Yaskawa INFORM job: DEMO_ROOF_SIDE_0625_3PAINT_28.JBI

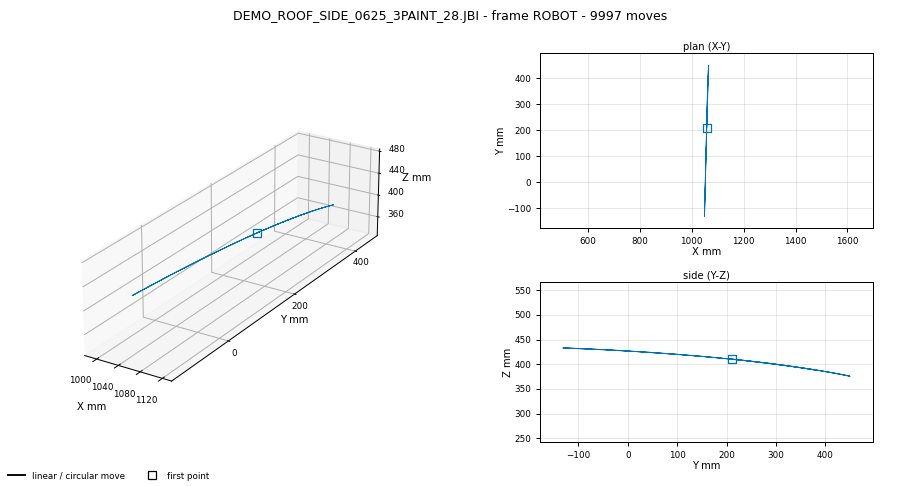
[picture p0: tool path of DEMO_ROOF_SIDE_0625_3PAINT_28.JBI in frame ROBOT, 9997 of 9997 moves have a stored position in this frame; points joined in program order, loops and branches not executed]
/JOB
//NAME DEMO_ROOF_SIDE_0625_3PAINT28
//POS
///NPOS 9997,0,0,0,0,0
///TOOL 0
///USER 0
///POSTYPE ROBOT
///RECTAN
///RCONF 1,0,0,0,0,0,0,0,0,0,0,0,0,0,0,0,0,0,0,0,0,0,0,0
C00000=1058.658,210.851,410.798,172.512,33.168,156.167
C00001=1058.665,211.100,410.772,172.514,33.173,156.168
C00002=1058.671,211.349,410.746,172.516,33.176,156.168
C00003=1058.677,211.597,410.720,172.518,33.181,156.169
C00004=1058.683,211.846,410.694,172.520,33.184,156.170
C00005=1058.690,212.094,410.668,172.522,33.189,156.171
C00006=1058.695,212.343,410.642,172.524,33.192,156.171
C00007=1058.702,212.591,410.616,172.526,33.196,156.172
C00008=1058.708,212.840,410.590,172.528,33.200,156.173
C00009=1058.714,213.088,410.564,172.530,33.204,156.174
C00010=1058.721,213.337,410.539,172.531,33.208,156.174
C00011=1058.726,213.585,410.512,172.533,33.212,156.175
C00012=1058.733,213.834,410.487,172.535,33.216,156.176
C00013=1058.738,214.082,410.460,172.537,33.220,156.177
C00014=1058.745,214.331,410.435,172.539,33.224,156.177
C00015=1058.751,214.580,410.408,172.541,33.227,156.178
C00016=1058.759,214.908,410.373,172.544,33.233,156.179
C00017=1058.767,215.238,410.338,172.546,33.238,156.180
C00018=1058.775,215.566,410.304,172.549,33.243,156.181
C00019=1058.783,215.895,410.269,172.553,33.248,156.182
C00020=1058.789,216.144,410.244,172.555,33.253,156.183
C00021=1058.795,216.392,410.217,172.557,33.256,156.184
C00022=1058.802,216.641,410.190,172.559,33.260,156.184
C00023=1058.808,216.890,410.165,172.561,33.264,156.185
C00024=1058.814,217.138,410.138,172.563,33.268,156.186
C00025=1058.820,217.386,410.112,172.565,33.271,156.186
C00026=1058.827,217.636,410.086,172.567,33.276,156.187
C00027=1058.832,217.884,410.059,172.569,33.279,156.188
C00028=1058.839,218.132,410.033,172.571,33.284,156.189
C00029=1058.845,218.380,410.007,172.573,33.287,156.189
C00030=1058.851,218.630,409.981,172.575,33.291,156.190
C00031=1058.857,218.878,409.954,172.577,33.295,156.191
C00032=1058.864,219.126,409.928,172.579,33.299,156.192
C00033=1058.870,219.375,409.901,172.581,33.302,156.192
C00034=1058.876,219.624,409.875,172.583,33.307,156.193
C00035=1058.882,219.872,409.849,172.585,33.310,156.194
C00036=1058.888,220.121,409.823,172.587,33.314,156.194
C00037=1058.895,220.369,409.796,172.589,33.318,156.195
C00038=1058.901,220.618,409.770,172.591,33.322,156.196
C00039=1058.907,220.866,409.744,172.593,33.326,156.197
C00040=1058.914,221.102,409.718,172.595,33.329,156.197
C00041=1058.918,221.337,409.693,172.598,33.333,156.198
C00042=1058.925,221.573,409.667,172.600,33.337,156.199
C00043=1058.930,221.809,409.643,172.601,33.340,156.199
C00044=1058.936,222.045,409.618,172.603,33.344,156.200
C00045=1058.942,222.280,409.593,172.605,33.348,156.201
C00046=1058.948,222.516,409.567,172.607,33.351,156.202
C00047=1058.954,222.752,409.542,172.609,33.355,156.202
C00048=1058.959,223.000,409.515,172.611,33.359,156.203
C00049=1058.966,223.249,409.488,172.613,33.363,156.204
C00050=1058.972,223.498,409.462,172.615,33.367,156.205
C00051=1058.977,223.746,409.435,172.617,33.371,156.205
C00052=1058.985,223.995,409.409,172.619,33.374,156.206
C00053=1058.990,224.243,409.382,172.621,33.379,156.207
C00054=1058.996,224.491,409.355,172.623,33.382,156.207
C00055=1059.003,224.740,409.328,172.626,33.386,156.208
C00056=1059.009,224.988,409.301,172.628,33.390,156.209
C00057=1059.016,225.237,409.275,172.630,33.394,156.210
C00058=1059.021,225.485,409.248,172.632,33.397,156.210
C00059=1059.027,225.734,409.221,172.635,33.402,156.211
C00060=1059.034,225.983,409.194,172.637,33.405,156.212
C00061=1059.039,226.231,409.168,172.639,33.409,156.212
C00062=1059.045,226.479,409.141,172.641,33.413,156.213
C00063=1059.053,226.728,409.114,172.643,33.417,156.214
C00064=1059.058,226.976,409.087,172.645,33.421,156.215
C00065=1059.065,227.225,409.060,172.647,33.424,156.215
C00066=1059.070,227.473,409.034,172.649,33.428,156.216
C00067=1059.077,227.722,409.007,172.651,33.432,156.217
C00068=1059.083,227.970,408.979,172.654,33.436,156.218
C00069=1059.090,228.219,408.953,172.656,33.439,156.218
C00070=1059.096,228.467,408.926,172.658,33.444,156.219
C00071=1059.102,228.716,408.899,172.660,33.447,156.220
C00072=1059.108,228.964,408.872,172.662,33.451,156.220
C00073=1059.114,229.212,408.845,172.664,33.455,156.221
C00074=1059.120,229.461,408.818,172.666,33.459,156.222
C00075=1059.126,229.710,408.791,172.669,33.463,156.223
C00076=1059.133,229.958,408.764,172.671,33.466,156.223
C00077=1059.139,230.207,408.737,172.673,33.470,156.224
C00078=1059.145,230.456,408.710,172.676,33.474,156.225
C00079=1059.151,230.703,408.683,172.678,33.478,156.226
C00080=1059.157,230.952,408.656,172.680,33.482,156.226
C00081=1059.164,231.200,408.628,172.682,33.486,156.227
C00082=1059.170,231.449,408.601,172.684,33.489,156.228
C00083=1059.176,231.698,408.575,172.686,33.494,156.229
C00084=1059.182,231.946,408.547,172.688,33.497,156.229
C00085=1059.188,232.194,408.520,172.690,33.501,156.230
C00086=1059.194,232.443,408.492,172.693,33.505,156.231
C00087=1059.200,232.692,408.465,172.695,33.509,156.231
C00088=1059.207,232.940,408.438,172.697,33.512,156.232
C00089=1059.212,233.188,408.411,172.700,33.516,156.233
C00090=1059.219,233.437,408.383,172.702,33.520,156.234
C00091=1059.225,233.685,408.357,172.704,33.524,156.234
C00092=1059.231,233.934,408.329,172.706,33.528,156.235
C00093=1059.236,234.182,408.302,172.708,33.532,156.236
C00094=1059.243,234.431,408.274,172.711,33.536,156.237
C00095=1059.249,234.679,408.247,172.713,33.539,156.237
C00096=1059.255,234.911,408.221,172.715,33.543,156.238
C00097=1059.261,235.142,408.196,172.717,33.546,156.239
C00098=1059.266,235.375,408.170,172.719,33.550,156.239
C00099=1059.272,235.606,408.144,172.721,33.554,156.240
C00100=1059.278,235.838,408.119,172.723,33.557,156.241
C00101=1059.284,236.070,408.093,172.725,33.560,156.241
C00102=1059.290,236.301,408.068,172.728,33.564,156.242
C00103=1059.295,236.532,408.042,172.730,33.568,156.243
C00104=1059.301,236.782,408.015,172.732,33.571,156.243
C00105=1059.307,237.030,407.987,172.734,33.576,156.244
C00106=1059.314,237.278,407.959,172.736,33.579,156.245
C00107=1059.320,237.527,407.932,172.739,33.583,156.246
C00108=1059.325,237.775,407.904,172.741,33.587,156.246
C00109=1059.332,238.023,407.877,172.743,33.591,156.247
C00110=1059.339,238.272,407.849,172.745,33.594,156.248
C00111=1059.344,238.520,407.822,172.747,33.598,156.248
C00112=1059.350,238.769,407.794,172.750,33.602,156.249
C00113=1059.357,239.017,407.766,172.752,33.606,156.250
C00114=1059.363,239.265,407.739,172.755,33.610,156.251
C00115=1059.370,239.514,407.711,172.757,33.613,156.251
C00116=1059.375,239.763,407.684,172.759,33.617,156.252
C00117=1059.382,240.011,407.656,172.762,33.621,156.253
C00118=1059.388,240.259,407.628,172.764,33.625,156.254
C00119=1059.394,240.508,407.600,172.766,33.628,156.254
C00120=1059.400,240.756,407.573,172.768,33.632,156.255
C00121=1059.407,241.004,407.545,172.770,33.636,156.256
C00122=1059.413,241.253,407.517,172.773,33.640,156.256
C00123=1059.419,241.501,407.490,172.775,33.644,156.257
C00124=1059.425,241.750,407.462,172.777,33.647,156.258
C00125=1059.431,241.998,407.434,172.780,33.651,156.259
C00126=1059.437,242.246,407.407,172.783,33.655,156.259
C00127=1059.443,242.495,407.378,172.785,33.659,156.260
C00128=1059.450,242.743,407.351,172.787,33.662,156.261
C00129=1059.455,242.991,407.323,172.789,33.666,156.261
C00130=1059.462,243.240,407.295,172.791,33.670,156.262
C00131=1059.468,243.489,407.267,172.794,33.674,156.263
C00132=1059.475,243.737,407.239,172.796,33.678,156.264
C00133=1059.480,243.985,407.211,172.798,33.682,156.265
C00134=1059.487,244.234,407.183,172.800,33.685,156.265
C00135=1059.493,244.482,407.155,172.803,33.689,156.266
C00136=1059.498,244.730,407.126,172.806,33.693,156.267
C00137=1059.505,244.978,407.098,172.808,33.697,156.267
C00138=1059.511,245.227,407.070,172.810,33.701,156.268
C00139=1059.517,245.475,407.042,172.813,33.704,156.269
C00140=1059.523,245.723,407.014,172.815,33.708,156.270
C00141=1059.530,245.972,406.987,172.817,33.712,156.270
C00142=1059.535,246.221,406.958,172.819,33.716,156.271
C00143=1059.542,246.469,406.929,172.822,33.719,156.272
C00144=1059.547,246.717,406.901,172.824,33.724,156.273
C00145=1059.554,246.965,406.874,172.826,33.727,156.273
C00146=1059.560,247.214,406.845,172.829,33.731,156.274
C00147=1059.566,247.463,406.817,172.832,33.735,156.275
C00148=1059.571,247.710,406.788,172.834,33.739,156.275
C00149=1059.578,247.959,406.761,172.836,33.743,156.276
C00150=1059.584,248.207,406.732,172.839,33.747,156.277
C00151=1059.590,248.456,406.703,172.841,33.750,156.278
C00152=1059.595,248.684,406.677,172.843,33.754,156.278
C00153=1059.601,248.913,406.652,172.845,33.757,156.279
C00154=1059.607,249.142,406.625,172.847,33.761,156.280
C00155=1059.611,249.370,406.599,172.850,33.765,156.280
C00156=1059.618,249.599,406.573,172.852,33.768,156.281
C00157=1059.623,249.828,406.547,172.854,33.771,156.282
C00158=1059.629,250.057,406.521,172.857,33.775,156.282
C00159=1059.634,250.285,406.495,172.859,33.779,156.283
C00160=1059.640,250.534,406.466,172.861,33.782,156.284
C00161=1059.647,250.782,406.437,172.863,33.786,156.285
C00162=1059.653,251.030,406.409,172.866,33.790,156.285
C00163=1059.659,251.278,406.380,172.868,33.794,156.286
C00164=1059.665,251.526,406.353,172.870,33.797,156.287
C00165=1059.671,251.774,406.323,172.873,33.802,156.288
C00166=1059.677,252.023,406.295,172.876,33.805,156.288
C00167=1059.683,252.271,406.266,172.878,33.809,156.289
C00168=1059.689,252.520,406.238,172.880,33.812,156.290
C00169=1059.695,252.768,406.209,172.883,33.817,156.291
C00170=1059.702,253.017,406.181,172.885,33.820,156.291
C00171=1059.708,253.265,406.152,172.887,33.824,156.292
C00172=1059.714,253.513,406.124,172.890,33.828,156.293
C00173=1059.720,253.761,406.095,172.893,33.832,156.293
C00174=1059.726,254.009,406.066,172.895,33.835,156.294
C00175=1059.732,254.258,406.038,172.898,33.839,156.295
C00176=1059.738,254.506,406.009,172.900,33.843,156.296
C00177=1059.745,254.754,405.981,172.903,33.847,156.296
C00178=1059.751,255.003,405.952,172.905,33.851,156.297
C00179=1059.758,255.251,405.923,172.907,33.854,156.298
C00180=1059.764,255.499,405.894,172.910,33.858,156.299
C00181=1059.770,255.748,405.865,172.912,33.862,156.299
C00182=1059.776,255.996,405.836,172.915,33.866,156.300
C00183=1059.782,256.244,405.808,172.918,33.869,156.301
C00184=1059.788,256.493,405.779,172.920,33.874,156.302
C00185=1059.794,256.741,405.750,172.922,33.877,156.302
C00186=1059.801,256.989,405.721,172.925,33.881,156.303
C00187=1059.807,257.237,405.693,172.927,33.884,156.304
C00188=1059.814,257.485,405.664,172.930,33.888,156.304
C00189=1059.820,257.734,405.635,172.932,33.892,156.305
C00190=1059.826,257.982,405.606,172.935,33.896,156.306
C00191=1059.832,258.230,405.578,172.938,33.900,156.307
C00192=1059.838,258.479,405.549,172.940,33.903,156.307
C00193=1059.845,258.727,405.520,172.943,33.907,156.308
C00194=1059.851,258.975,405.491,172.945,33.911,156.309
C00195=1059.857,259.223,405.462,172.947,33.915,156.309
C00196=1059.863,259.471,405.433,172.950,33.918,156.310
C00197=1059.869,259.720,405.404,172.952,33.922,156.311
C00198=1059.876,259.968,405.375,172.956,33.926,156.312
C00199=1059.883,260.216,405.347,172.958,33.930,156.312
C00200=1059.889,260.465,405.317,172.961,33.933,156.313
C00201=1059.896,260.713,405.288,172.963,33.937,156.314
C00202=1059.902,260.961,405.259,172.965,33.941,156.315
C00203=1059.908,261.209,405.230,172.968,33.944,156.315
C00204=1059.914,261.457,405.201,172.970,33.948,156.316
C00205=1059.921,261.705,405.172,172.973,33.952,156.317
C00206=1059.927,261.953,405.143,172.976,33.956,156.317
C00207=1059.933,262.202,405.114,172.979,33.959,156.318
C00208=1059.939,262.430,405.087,172.981,33.963,156.319
C00209=1059.945,262.657,405.060,172.983,33.966,156.319
C00210=1059.951,262.885,405.034,172.985,33.970,156.320
C00211=1059.957,263.113,405.007,172.988,33.973,156.321
C00212=1059.963,263.340,404.981,172.990,33.976,156.321
C00213=1059.968,263.568,404.954,172.992,33.980,156.322
C00214=1059.974,263.796,404.927,172.995,33.983,156.323
C00215=1059.979,264.023,404.899,172.998,33.987,156.324
C00216=1059.985,264.271,404.870,173.000,33.991,156.324
C00217=1059.992,264.519,404.841,173.002,33.995,156.325
C00218=1059.998,264.768,404.812,173.005,33.999,156.326
C00219=1060.003,265.016,404.782,173.007,34.002,156.326
C00220=1060.010,265.265,404.753,173.010,34.006,156.327
C00221=1060.017,265.512,404.723,173.013,34.010,156.328
C00222=1060.022,265.761,404.693,173.016,34.014,156.329
C00223=1060.029,266.009,404.664,173.018,34.017,156.329
C00224=1060.035,266.257,404.635,173.021,34.021,156.330
C00225=1060.041,266.505,404.605,173.023,34.025,156.331
C00226=1060.048,266.754,404.576,173.026,34.029,156.332
C00227=1060.054,267.002,404.547,173.028,34.033,156.332
C00228=1060.060,267.250,404.516,173.032,34.036,156.333
C00229=1060.066,267.498,404.487,173.034,34.040,156.334
C00230=1060.072,267.746,404.458,173.037,34.044,156.335
C00231=1060.079,267.994,404.428,173.039,34.048,156.335
C00232=1060.085,268.243,404.398,173.042,34.052,156.336
C00233=1060.091,268.491,404.369,173.044,34.055,156.337
C00234=1060.097,268.739,404.339,173.047,34.059,156.338
C00235=1060.103,268.987,404.310,173.050,34.063,156.338
C00236=1060.110,269.235,404.280,173.053,34.067,156.339
C00237=1060.116,269.483,404.250,173.055,34.071,156.340
C00238=1060.122,269.731,404.220,173.058,34.074,156.341
C00239=1060.128,269.979,404.191,173.060,34.079,156.341
C00240=1060.135,270.227,404.161,173.063,34.082,156.342
C00241=1060.141,270.476,404.131,173.065,34.086,156.343
C00242=1060.147,270.723,404.101,173.069,34.090,156.344
C00243=1060.153,270.972,404.072,173.071,34.094,156.344
C00244=1060.160,271.220,404.042,173.074,34.097,156.345
C00245=1060.165,271.469,404.012,173.076,34.101,156.346
C00246=1060.172,271.716,403.982,173.079,34.105,156.347
C00247=1060.178,271.965,403.952,173.081,34.109,156.347
C00248=1060.184,272.213,403.922,173.085,34.113,156.348
C00249=1060.190,272.461,403.892,173.087,34.116,156.349
C00250=1060.197,272.709,403.863,173.090,34.120,156.350
C00251=1060.203,272.957,403.832,173.092,34.124,156.350
C00252=1060.210,273.205,403.802,173.095,34.128,156.351
C00253=1060.215,273.453,403.773,173.097,34.132,156.352
C00254=1060.221,273.702,403.742,173.101,34.136,156.353
C00255=1060.228,273.949,403.712,173.104,34.139,156.353
C00256=1060.234,274.198,403.683,173.106,34.143,156.354
C00257=1060.240,274.446,403.652,173.109,34.147,156.355
C00258=1060.247,274.694,403.622,173.111,34.151,156.356
C00259=1060.252,274.941,403.592,173.114,34.155,156.356
C00260=1060.258,275.191,403.562,173.116,34.158,156.357
C00261=1060.265,275.438,403.532,173.120,34.163,156.358
C00262=1060.271,275.686,403.502,173.123,34.166,156.359
C00263=1060.277,275.934,403.471,173.125,34.170,156.360
C00264=1060.284,276.164,403.443,173.127,34.174,156.360
C00265=1060.289,276.394,403.416,173.130,34.178,156.361
C00266=1060.295,276.623,403.388,173.132,34.181,156.362
C00267=1060.300,276.852,403.360,173.136,34.184,156.362
C00268=1060.306,277.082,403.331,173.138,34.188,156.363
C00269=1060.311,277.312,403.304,173.140,34.191,156.364
C00270=1060.317,277.541,403.276,173.143,34.195,156.364
C00271=1060.323,277.771,403.247,173.145,34.199,156.365
C00272=1060.330,278.019,403.217,173.148,34.203,156.366
C00273=1060.336,278.266,403.187,173.151,34.206,156.367
C00274=1060.342,278.515,403.156,173.154,34.211,156.367
C00275=1060.348,278.763,403.126,173.157,34.214,156.368
C00276=1060.355,279.011,403.096,173.159,34.218,156.369
C00277=1060.361,279.259,403.065,173.162,34.222,156.370
C00278=1060.367,279.507,403.035,173.165,34.226,156.370
C00279=1060.373,279.755,403.004,173.168,34.230,156.371
C00280=1060.380,280.003,402.974,173.171,34.233,156.372
C00281=1060.386,280.251,402.944,173.173,34.237,156.373
C00282=1060.392,280.499,402.914,173.176,34.241,156.374
C00283=1060.398,280.748,402.883,173.179,34.245,156.374
C00284=1060.404,280.995,402.853,173.181,34.249,156.375
C00285=1060.411,281.243,402.821,173.185,34.253,156.376
C00286=1060.417,281.491,402.791,173.187,34.257,156.377
C00287=1060.423,281.740,402.760,173.190,34.261,156.377
C00288=1060.429,281.987,402.730,173.193,34.264,156.378
C00289=1060.435,282.236,402.699,173.195,34.269,156.379
C00290=1060.442,282.483,402.668,173.199,34.272,156.380
C00291=1060.448,282.732,402.637,173.202,34.276,156.381
C00292=1060.454,282.979,402.607,173.204,34.280,156.381
C00293=1060.460,283.228,402.576,173.207,34.284,156.382
C00294=1060.466,283.475,402.545,173.210,34.288,156.383
C00295=1060.473,283.724,402.514,173.213,34.292,156.384
C00296=1060.479,283.972,402.484,173.216,34.296,156.384
C00297=1060.485,284.219,402.453,173.219,34.300,156.385
C00298=1060.491,284.467,402.422,173.221,34.304,156.386
C00299=1060.498,284.716,402.391,173.224,34.307,156.387
C00300=1060.504,284.963,402.360,173.227,34.312,156.388
C00301=1060.510,285.212,402.330,173.230,34.315,156.388
C00302=1060.517,285.459,402.298,173.233,34.319,156.389
C00303=1060.523,285.707,402.268,173.236,34.323,156.390
C00304=1060.529,285.956,402.237,173.238,34.327,156.391
C00305=1060.535,286.203,402.206,173.241,34.331,156.391
C00306=1060.542,286.451,402.175,173.245,34.335,156.392
C00307=1060.548,286.699,402.144,173.247,34.338,156.393
C00308=1060.554,286.947,402.114,173.250,34.343,156.394
C00309=1060.561,287.195,402.082,173.253,34.347,156.395
C00310=1060.567,287.444,402.051,173.256,34.350,156.395
C00311=1060.573,287.691,402.020,173.259,34.355,156.396
C00312=1060.580,287.939,401.990,173.262,34.358,156.397
C00313=1060.587,288.187,401.958,173.265,34.362,156.398
C00314=1060.592,288.435,401.927,173.267,34.366,156.398
C00315=1060.598,288.683,401.896,173.270,34.370,156.399
C00316=1060.604,288.930,401.865,173.274,34.374,156.400
C00317=1060.611,289.179,401.834,173.277,34.378,156.401
C00318=1060.618,289.427,401.803,173.279,34.382,156.402
C00319=1060.623,289.674,401.771,173.282,34.386,156.402
C00320=1060.629,289.910,401.742,173.285,34.390,156.403
C00321=1060.636,290.145,401.712,173.288,34.393,156.404
C00322=1060.641,290.380,401.683,173.291,34.397,156.405
C00323=1060.647,290.615,401.653,173.293,34.401,156.405
C00324=1060.653,290.850,401.623,173.296,34.405,156.406
C00325=1060.659,291.084,401.594,173.299,34.408,156.407
C00326=1060.665,291.320,401.563,173.302,34.412,156.408
C00327=1060.671,291.555,401.534,173.305,34.416,156.408
C00328=1060.677,291.802,401.503,173.308,34.420,156.409
C00329=1060.683,292.050,401.471,173.310,34.424,156.410
C00330=1060.690,292.298,401.440,173.313,34.428,156.411
C00331=1060.697,292.546,401.408,173.317,34.432,156.412
C00332=1060.702,292.794,401.377,173.320,34.436,156.412
C00333=1060.709,293.042,401.345,173.322,34.440,156.413
C00334=1060.715,293.290,401.315,173.325,34.444,156.414
C00335=1060.721,293.538,401.283,173.328,34.447,156.415
C00336=1060.727,293.786,401.252,173.332,34.452,156.416
C00337=1060.734,294.033,401.220,173.335,34.456,156.416
C00338=1060.740,294.282,401.188,173.337,34.459,156.417
C00339=1060.747,294.530,401.157,173.340,34.463,156.418
C00340=1060.753,294.777,401.126,173.344,34.468,156.419
C00341=1060.759,295.025,401.094,173.347,34.472,156.420
C00342=1060.765,295.273,401.062,173.350,34.475,156.420
C00343=1060.771,295.521,401.030,173.352,34.479,156.421
C00344=1060.778,295.769,400.999,173.355,34.484,156.422
C00345=1060.784,296.017,400.967,173.359,34.488,156.423
C00346=1060.790,296.264,400.936,173.362,34.491,156.424
C00347=1060.796,296.513,400.904,173.365,34.495,156.425
C00348=1060.803,296.760,400.871,173.367,34.500,156.425
C00349=1060.809,297.008,400.839,173.371,34.504,156.426
C00350=1060.815,297.255,400.808,173.374,34.508,156.427
C00351=1060.821,297.504,400.776,173.377,34.512,156.428
C00352=1060.827,297.752,400.744,173.380,34.516,156.429
C00353=1060.834,297.999,400.712,173.382,34.520,156.429
C00354=1060.840,298.247,400.680,173.386,34.524,156.430
C00355=1060.846,298.495,400.648,173.389,34.528,156.431
C00356=1060.852,298.743,400.616,173.392,34.532,156.432
C00357=1060.859,298.990,400.584,173.395,34.536,156.433
C00358=1060.865,299.238,400.552,173.399,34.540,156.434
C00359=1060.871,299.487,400.520,173.401,34.545,156.435
C00360=1060.877,299.734,400.487,173.404,34.549,156.435
C00361=1060.883,299.981,400.456,173.407,34.553,156.436
C00362=1060.889,300.230,400.424,173.411,34.557,156.437
C00363=1060.895,300.477,400.392,173.414,34.561,156.438
C00364=1060.901,300.725,400.360,173.417,34.565,156.439
C00365=1060.908,300.973,400.327,173.419,34.569,156.440
C00366=1060.915,301.221,400.295,173.423,34.574,156.440
C00367=1060.920,301.469,400.263,173.426,34.578,156.441
C00368=1060.927,301.717,400.231,173.429,34.582,156.442
C00369=1060.932,301.964,400.199,173.432,34.586,156.443
C00370=1060.938,302.212,400.166,173.436,34.590,156.444
C00371=1060.945,302.460,400.135,173.439,34.594,156.445
C00372=1060.951,302.707,400.102,173.441,34.598,156.445
C00373=1060.958,302.955,400.069,173.444,34.602,156.446
C00374=1060.964,303.203,400.037,173.448,34.607,156.447
C00375=1060.970,303.451,400.005,173.451,34.611,156.448
C00376=1060.977,303.693,399.974,173.454,34.615,156.449
C00377=1060.983,303.936,399.942,173.457,34.618,156.450
C00378=1060.989,304.178,399.910,173.460,34.623,156.450
C00379=1060.995,304.421,399.878,173.464,34.627,156.451
C00380=1061.001,304.664,399.847,173.466,34.631,156.452
C00381=1061.007,304.906,399.815,173.469,34.635,156.453
C00382=1061.013,305.149,399.783,173.473,34.639,156.454
C00383=1061.019,305.392,399.752,173.476,34.643,156.455
C00384=1061.026,305.639,399.719,173.479,34.647,156.456
C00385=1061.033,305.887,399.687,173.482,34.651,156.456
C00386=1061.039,306.135,399.654,173.486,34.656,156.457
C00387=1061.045,306.383,399.622,173.489,34.660,156.458
C00388=1061.051,306.630,399.589,173.492,34.664,156.459
C00389=1061.058,306.878,399.556,173.495,34.668,156.460
C00390=1061.064,307.126,399.523,173.499,34.672,156.461
C00391=1061.071,307.374,399.491,173.502,34.676,156.461
C00392=1061.077,307.622,399.459,173.504,34.680,156.462
C00393=1061.084,307.869,399.426,173.507,34.684,156.463
C00394=1061.090,308.117,399.394,173.511,34.689,156.464
C00395=1061.096,308.364,399.361,173.514,34.693,156.465
C00396=1061.103,308.612,399.328,173.517,34.697,156.466
C00397=1061.109,308.860,399.295,173.520,34.701,156.467
C00398=1061.116,309.108,399.262,173.524,34.705,156.467
C00399=1061.123,309.355,399.230,173.527,34.709,156.468
C00400=1061.129,309.603,399.197,173.530,34.713,156.469
C00401=1061.135,309.850,399.165,173.533,34.717,156.470
C00402=1061.141,310.099,399.133,173.537,34.722,156.471
C00403=1061.148,310.347,399.100,173.540,34.726,156.472
C00404=1061.155,310.595,399.067,173.543,34.730,156.473
C00405=1061.161,310.842,399.033,173.547,34.734,156.473
C00406=1061.167,311.089,399.001,173.550,34.739,156.474
C00407=1061.174,311.337,398.968,173.553,34.743,156.475
C00408=1061.181,311.585,398.935,173.556,34.747,156.476
C00409=1061.187,311.833,398.902,173.560,34.751,156.477
C00410=1061.193,312.080,398.869,173.563,34.755,156.478
C00411=1061.200,312.328,398.836,173.566,34.759,156.479
C00412=1061.207,312.576,398.804,173.570,34.764,156.480
C00413=1061.213,312.823,398.771,173.573,34.768,156.480
C00414=1061.220,313.072,398.738,173.576,34.772,156.481
C00415=1061.227,313.319,398.705,173.580,34.776,156.482
C00416=1061.233,313.566,398.672,173.584,34.780,156.483
C00417=1061.240,313.815,398.639,173.587,34.784,156.484
C00418=1061.246,314.062,398.606,173.590,34.789,156.485
C00419=1061.252,314.309,398.572,173.593,34.793,156.486
C00420=1061.258,314.557,398.539,173.597,34.798,156.487
C00421=1061.265,314.806,398.506,173.600,34.802,156.487
C00422=1061.271,315.053,398.472,173.603,34.807,156.488
C00423=1061.277,315.300,398.439,173.607,34.811,156.489
C00424=1061.283,315.548,398.406,173.610,34.815,156.490
C00425=1061.290,315.796,398.372,173.613,34.820,156.491
C00426=1061.296,316.044,398.339,173.617,34.824,156.492
C00427=1061.302,316.291,398.305,173.620,34.828,156.493
C00428=1061.309,316.539,398.272,173.623,34.832,156.494
C00429=1061.315,316.786,398.238,173.627,34.837,156.495
C00430=1061.321,317.034,398.205,173.630,34.841,156.496
C00431=1061.327,317.282,398.171,173.633,34.846,156.497
C00432=1061.333,317.526,398.138,173.636,34.850,156.497
C00433=1061.340,317.771,398.105,173.640,34.855,156.498
C00434=1061.345,318.015,398.072,173.643,34.859,156.499
C00435=1061.352,318.260,398.039,173.646,34.863,156.500
C00436=1061.359,318.504,398.005,173.650,34.867,156.501
C00437=1061.365,318.749,397.973,173.653,34.872,156.502
C00438=1061.371,318.994,397.939,173.656,34.876,156.503
C00439=1061.377,319.238,397.906,173.660,34.880,156.504
C00440=1061.383,319.485,397.872,173.663,34.885,156.505
C00441=1061.390,319.733,397.838,173.666,34.889,156.506
C00442=1061.396,319.981,397.805,173.671,34.894,156.507
C00443=1061.403,320.229,397.771,173.674,34.898,156.508
C00444=1061.409,320.476,397.737,173.677,34.902,156.508
C00445=1061.416,320.724,397.703,173.681,34.907,156.509
C00446=1061.422,320.972,397.670,173.684,34.911,156.510
C00447=1061.429,321.219,397.636,173.687,34.916,156.511
C00448=1061.435,321.466,397.602,173.691,34.921,156.512
C00449=1061.442,321.714,397.568,173.694,34.925,156.513
C00450=1061.447,321.962,397.535,173.697,34.929,156.514
C00451=1061.454,322.210,397.501,173.701,34.933,156.515
C00452=1061.460,322.457,397.467,173.705,34.938,156.516
C00453=1061.467,322.705,397.433,173.708,34.943,156.517
C00454=1061.474,322.952,397.399,173.711,34.947,156.518
C00455=1061.480,323.200,397.365,173.715,34.951,156.519
C00456=1061.487,323.447,397.331,173.718,34.956,156.520
C00457=1061.493,323.695,397.297,173.721,34.960,156.521
C00458=1061.499,323.944,397.263,173.726,34.965,156.522
C00459=1061.506,324.191,397.230,173.729,34.969,156.523
C00460=1061.512,324.439,397.195,173.732,34.974,156.523
C00461=1061.519,324.685,397.162,173.736,34.978,156.524
C00462=1061.525,324.933,397.127,173.739,34.983,156.525
C00463=1061.532,325.181,397.093,173.742,34.987,156.526
C00464=1061.538,325.428,397.060,173.747,34.992,156.527
C00465=1061.545,325.676,397.024,173.750,34.996,156.528
C00466=1061.552,325.923,396.991,173.754,35.001,156.529
C00467=1061.558,326.171,396.957,173.757,35.005,156.530
C00468=1061.565,326.419,396.922,173.760,35.010,156.531
C00469=1061.572,326.666,396.888,173.765,35.014,156.532
C00470=1061.578,326.914,396.854,173.768,35.019,156.533
C00471=1061.585,327.161,396.820,173.771,35.023,156.534
C00472=1061.591,327.409,396.786,173.775,35.028,156.535
C00473=1061.598,327.657,396.751,173.779,35.032,156.536
C00474=1061.605,327.904,396.717,173.782,35.037,156.537
C00475=1061.611,328.152,396.683,173.786,35.041,156.538
C00476=1061.618,328.400,396.649,173.789,35.046,156.539
C00477=1061.625,328.647,396.614,173.792,35.050,156.540
C00478=1061.631,328.894,396.580,173.797,35.055,156.541
C00479=1061.638,329.142,396.546,173.800,35.059,156.542
C00480=1061.645,329.390,396.512,173.803,35.064,156.543
C00481=1061.651,329.637,396.477,173.807,35.068,156.544
C00482=1061.658,329.885,396.442,173.811,35.073,156.545
C00483=1061.665,330.132,396.409,173.815,35.077,156.546
C00484=1061.671,330.379,396.374,173.818,35.082,156.547
C00485=1061.678,330.627,396.339,173.822,35.087,156.547
C00486=1061.685,330.875,396.304,173.826,35.091,156.548
C00487=1061.691,331.123,396.270,173.829,35.096,156.549
C00488=1061.697,331.364,396.235,173.832,35.101,156.550
C00489=1061.704,331.606,396.202,173.836,35.105,156.551
C00490=1061.710,331.847,396.168,173.840,35.110,156.552
C00491=1061.716,332.089,396.134,173.844,35.114,156.553
C00492=1061.723,332.331,396.100,173.847,35.119,156.554
C00493=1061.729,332.572,396.066,173.850,35.124,156.555
C00494=1061.735,332.814,396.033,173.854,35.128,156.556
C00495=1061.742,333.056,395.998,173.858,35.133,156.557
C00496=1061.749,333.303,395.963,173.861,35.138,156.558
C00497=1061.755,333.550,395.929,173.865,35.142,156.559
C00498=1061.762,333.798,395.894,173.869,35.147,156.560
C00499=1061.768,334.045,395.859,173.873,35.151,156.561
C00500=1061.775,334.293,395.824,173.876,35.157,156.562
C00501=1061.781,334.541,395.789,173.879,35.161,156.563
C00502=1061.788,334.788,395.753,173.884,35.166,156.564
C00503=1061.794,335.035,395.718,173.887,35.170,156.565
C00504=1061.801,335.283,395.684,173.891,35.175,156.566
C00505=1061.808,335.531,395.649,173.895,35.180,156.568
C00506=1061.814,335.778,395.614,173.898,35.185,156.569
C00507=1061.821,336.026,395.578,173.902,35.189,156.570
C00508=1061.828,336.273,395.543,173.906,35.195,156.571
C00509=1061.834,336.520,395.509,173.910,35.199,156.572
C00510=1061.841,336.767,395.473,173.913,35.204,156.573
C00511=1061.848,337.014,395.438,173.917,35.208,156.574
C00512=1061.853,337.263,395.403,173.921,35.214,156.575
C00513=1061.860,337.510,395.368,173.925,35.218,156.576
C00514=1061.867,337.757,395.333,173.929,35.223,156.577
C00515=1061.873,338.004,395.297,173.932,35.228,156.578
C00516=1061.880,338.252,395.261,173.937,35.233,156.579
C00517=1061.887,338.499,395.226,173.940,35.238,156.580
C00518=1061.893,338.747,395.191,173.943,35.243,156.581
C00519=1061.900,338.994,395.155,173.948,35.248,156.582
C00520=1061.906,339.241,395.120,173.951,35.253,156.583
C00521=1061.913,339.489,395.085,173.956,35.257,156.584
C00522=1061.919,339.737,395.049,173.959,35.262,156.585
C00523=1061.926,339.984,395.014,173.962,35.267,156.586
C00524=1061.934,340.231,394.978,173.967,35.272,156.587
C00525=1061.940,340.479,394.942,173.970,35.277,156.588
C00526=1061.946,340.726,394.907,173.975,35.282,156.590
C00527=1061.953,340.974,394.872,173.978,35.287,156.591
C00528=1061.959,341.221,394.836,173.982,35.292,156.592
C00529=1061.966,341.468,394.800,173.986,35.297,156.593
C00530=1061.972,341.716,394.765,173.990,35.301,156.594
C00531=1061.979,341.963,394.730,173.994,35.307,156.595
C00532=1061.986,342.210,394.694,173.997,35.312,156.596
C00533=1061.993,342.458,394.658,174.002,35.316,156.597
C00534=1061.999,342.706,394.623,174.005,35.322,156.598
C00535=1062.007,342.952,394.587,174.009,35.327,156.599
C00536=1062.013,343.200,394.551,174.013,35.331,156.600
C00537=1062.020,343.447,394.515,174.017,35.336,156.601
C00538=1062.026,343.695,394.479,174.021,35.342,156.603
C00539=1062.033,343.942,394.443,174.025,35.347,156.604
C00540=1062.039,344.190,394.407,174.029,35.352,156.605
C00541=1062.046,344.436,394.372,174.033,35.357,156.606
C00542=1062.052,344.684,394.336,174.037,35.362,156.607
C00543=1062.059,344.931,394.299,174.041,35.367,156.608
C00544=1062.065,345.171,394.265,174.044,35.372,156.609
C00545=1062.072,345.410,394.230,174.048,35.377,156.610
C00546=1062.079,345.649,394.195,174.052,35.382,156.611
C00547=1062.085,345.888,394.160,174.056,35.387,156.613
C00548=1062.092,346.127,394.125,174.060,35.391,156.614
C00549=1062.098,346.367,394.091,174.063,35.396,156.615
C00550=1062.104,346.606,394.056,174.068,35.402,156.616
C00551=1062.111,346.846,394.021,174.071,35.407,156.617
C00552=1062.118,347.093,393.984,174.076,35.412,156.618
C00553=1062.125,347.340,393.948,174.079,35.417,156.619
C00554=1062.131,347.588,393.912,174.084,35.422,156.620
C00555=1062.137,347.835,393.876,174.087,35.427,156.621
C00556=1062.145,348.082,393.840,174.092,35.432,156.623
C00557=1062.151,348.329,393.803,174.095,35.437,156.624
C00558=1062.157,348.576,393.767,174.100,35.443,156.625
C00559=1062.165,348.824,393.730,174.103,35.448,156.626
C00560=1062.171,349.071,393.694,174.108,35.453,156.627
C00561=1062.177,349.319,393.658,174.111,35.458,156.628
C00562=1062.184,349.566,393.621,174.116,35.464,156.629
C00563=1062.191,349.813,393.586,174.120,35.469,156.631
C00564=1062.198,350.061,393.549,174.124,35.474,156.632
C00565=1062.205,350.308,393.512,174.128,35.479,156.633
C00566=1062.211,350.555,393.476,174.132,35.484,156.634
C00567=1062.219,350.802,393.440,174.136,35.490,156.635
C00568=1062.225,351.049,393.403,174.140,35.495,156.636
C00569=1062.232,351.297,393.366,174.144,35.500,156.638
C00570=1062.239,351.544,393.329,174.149,35.505,156.639
C00571=1062.246,351.791,393.293,174.152,35.511,156.640
C00572=1062.253,352.038,393.257,174.157,35.516,156.641
C00573=1062.259,352.285,393.220,174.160,35.522,156.642
C00574=1062.266,352.533,393.183,174.165,35.527,156.643
C00575=1062.273,352.779,393.146,174.169,35.532,156.645
C00576=1062.280,353.027,393.109,174.173,35.538,156.646
C00577=1062.286,353.274,393.073,174.177,35.543,156.647
C00578=1062.293,353.521,393.035,174.182,35.548,156.648
C00579=1062.299,353.768,392.999,174.186,35.554,156.650
C00580=1062.306,354.016,392.962,174.190,35.559,156.651
C00581=1062.313,354.263,392.925,174.194,35.565,156.652
C00582=1062.320,354.510,392.888,174.198,35.570,156.653
C00583=1062.326,354.757,392.852,174.203,35.576,156.654
C00584=1062.334,355.005,392.814,174.206,35.581,156.656
C00585=1062.340,355.252,392.778,174.211,35.586,156.657
C00586=1062.347,355.499,392.740,174.215,35.592,156.658
C00587=1062.353,355.746,392.704,174.219,35.597,156.659
C00588=1062.361,355.993,392.666,174.224,35.603,156.660
C00589=1062.368,356.241,392.629,174.228,35.608,156.662
C00590=1062.374,356.487,392.592,174.232,35.613,156.663
C00591=1062.381,356.735,392.556,174.236,35.619,156.664
C00592=1062.388,356.981,392.518,174.241,35.625,156.665
C00593=1062.395,357.228,392.481,174.244,35.630,156.667
C00594=1062.402,357.476,392.444,174.249,35.635,156.668
C00595=1062.409,357.723,392.407,174.254,35.641,156.669
C00596=1062.416,357.970,392.369,174.257,35.647,156.670
C00597=1062.423,358.218,392.333,174.262,35.652,156.672
C00598=1062.430,358.464,392.295,174.266,35.657,156.673
C00599=1062.436,358.711,392.257,174.271,35.663,156.674
C00600=1062.442,358.953,392.221,174.274,35.669,156.675
C00601=1062.450,359.195,392.184,174.279,35.674,156.677
C00602=1062.456,359.436,392.148,174.284,35.680,156.678
C00603=1062.463,359.677,392.111,174.287,35.685,156.679
C00604=1062.469,359.919,392.075,174.292,35.691,156.680
C00605=1062.476,360.161,392.038,174.295,35.696,156.682
C00606=1062.483,360.402,392.001,174.300,35.702,156.683
C00607=1062.490,360.643,391.965,174.305,35.708,156.684
C00608=1062.497,360.890,391.927,174.309,35.713,156.685
C00609=1062.504,361.137,391.890,174.313,35.719,156.687
C00610=1062.510,361.384,391.852,174.317,35.725,156.688
C00611=1062.517,361.631,391.814,174.322,35.730,156.689
C00612=1062.525,361.878,391.777,174.327,35.736,156.690
C00613=1062.532,362.125,391.739,174.330,35.741,156.692
C00614=1062.538,362.373,391.701,174.335,35.748,156.693
C00615=1062.545,362.619,391.664,174.340,35.753,156.694
C00616=1062.552,362.866,391.627,174.344,35.759,156.696
C00617=1062.559,363.114,391.588,174.349,35.764,156.697
C00618=1062.566,363.360,391.550,174.353,35.771,156.698
C00619=1062.574,363.607,391.513,174.357,35.776,156.700
C00620=1062.580,363.855,391.475,174.362,35.782,156.701
C00621=1062.587,364.102,391.437,174.366,35.788,156.702
C00622=1062.593,364.349,391.399,174.371,35.794,156.704
C00623=1062.601,364.595,391.361,174.375,35.800,156.705
C00624=1062.607,364.842,391.323,174.379,35.805,156.706
C00625=1062.615,365.090,391.285,174.384,35.812,156.708
C00626=1062.621,365.336,391.247,174.389,35.817,156.709
C00627=1062.629,365.584,391.209,174.393,35.823,156.710
C00628=1062.635,365.830,391.170,174.398,35.829,156.712
C00629=1062.642,366.077,391.133,174.402,35.835,156.713
C00630=1062.649,366.324,391.094,174.406,35.841,156.715
C00631=1062.656,366.571,391.057,174.411,35.847,156.716
C00632=1062.663,366.818,391.018,174.416,35.853,156.717
C00633=1062.669,367.065,390.980,174.420,35.859,156.719
C00634=1062.677,367.312,390.941,174.425,35.865,156.720
C00635=1062.684,367.559,390.903,174.430,35.871,156.721
C00636=1062.691,367.806,390.865,174.435,35.877,156.723
C00637=1062.698,368.052,390.826,174.438,35.883,156.724
C00638=1062.704,368.300,390.788,174.443,35.889,156.725
C00639=1062.712,368.546,390.750,174.448,35.895,156.727
C00640=1062.719,368.793,390.711,174.452,35.901,156.728
C00641=1062.726,369.040,390.673,174.457,35.907,156.730
C00642=1062.733,369.287,390.635,174.462,35.913,156.731
C00643=1062.740,369.534,390.596,174.466,35.919,156.733
C00644=1062.747,369.780,390.558,174.471,35.926,156.734
C00645=1062.754,370.027,390.519,174.476,35.932,156.735
C00646=1062.760,370.275,390.481,174.481,35.938,156.737
C00647=1062.769,370.522,390.442,174.485,35.944,156.738
C00648=1062.775,370.769,390.403,174.490,35.950,156.740
C00649=1062.783,371.015,390.365,174.495,35.956,156.741
C00650=1062.790,371.262,390.326,174.500,35.962,156.742
C00651=1062.797,371.509,390.287,174.504,35.969,156.744
C00652=1062.804,371.755,390.249,174.508,35.975,156.745
C00653=1062.811,372.002,390.210,174.513,35.981,156.747
C00654=1062.818,372.250,390.171,174.517,35.987,156.748
C00655=1062.826,372.496,390.133,174.522,35.993,156.750
C00656=1062.833,372.749,390.092,174.528,36.000,156.751
C00657=1062.840,373.004,390.052,174.533,36.006,156.752
C00658=1062.848,373.258,390.012,174.538,36.012,156.754
C00659=1062.854,373.511,389.973,174.542,36.019,156.756
C00660=1062.862,373.758,389.933,174.547,36.025,156.757
C00661=1062.868,374.005,389.894,174.552,36.032,156.759
C00662=1062.875,374.252,389.855,174.557,36.038,156.760
C00663=1062.882,374.499,389.816,174.562,36.045,156.762
C00664=1062.889,374.745,389.777,174.566,36.051,156.763
C00665=1062.897,374.993,389.738,174.571,36.057,156.765
C00666=1062.903,375.239,389.699,174.576,36.064,156.766
C00667=1062.911,375.486,389.659,174.581,36.070,156.768
C00668=1062.918,375.732,389.621,174.586,36.077,156.769
C00669=1062.926,375.979,389.581,174.590,36.083,156.770
C00670=1062.933,376.226,389.542,174.595,36.090,156.772
C00671=1062.940,376.472,389.503,174.600,36.096,156.774
C00672=1062.947,376.720,389.463,174.605,36.102,156.775
C00673=1062.954,376.966,389.424,174.610,36.109,156.777
C00674=1062.961,377.213,389.385,174.614,36.116,156.778
C00675=1062.969,377.460,389.345,174.620,36.122,156.780
C00676=1062.976,377.706,389.306,174.625,36.128,156.781
C00677=1062.983,377.953,389.267,174.630,36.135,156.783
C00678=1062.990,378.199,389.227,174.635,36.142,156.784
C00679=1062.997,378.446,389.188,174.640,36.148,156.786
C00680=1063.004,378.694,389.147,174.644,36.155,156.787
C00681=1063.011,378.940,389.108,174.649,36.162,156.789
C00682=1063.018,379.187,389.069,174.654,36.168,156.790
C00683=1063.026,379.433,389.029,174.659,36.175,156.792
C00684=1063.033,379.680,388.990,174.665,36.181,156.794
C00685=1063.041,379.927,388.950,174.670,36.188,156.795
C00686=1063.048,380.173,388.910,174.674,36.195,156.797
C00687=1063.055,380.420,388.871,174.679,36.201,156.798
C00688=1063.062,380.666,388.831,174.684,36.208,156.800
C00689=1063.070,380.913,388.791,174.689,36.215,156.801
C00690=1063.077,381.160,388.752,174.695,36.222,156.803
C00691=1063.084,381.407,388.711,174.700,36.228,156.805
C00692=1063.091,381.653,388.672,174.705,36.235,156.806
C00693=1063.099,381.900,388.632,174.710,36.242,156.808
C00694=1063.105,382.146,388.592,174.715,36.249,156.810
C00695=1063.113,382.393,388.551,174.721,36.256,156.811
C00696=1063.121,382.639,388.512,174.725,36.262,156.813
C00697=1063.128,382.886,388.471,174.730,36.270,156.814
C00698=1063.135,383.133,388.431,174.735,36.276,156.816
C00699=1063.142,383.379,388.392,174.740,36.283,156.818
C00700=1063.149,383.626,388.351,174.746,36.290,156.819
C00701=1063.157,383.872,388.311,174.751,36.297,156.821
C00702=1063.164,384.119,388.270,174.756,36.304,156.823
C00703=1063.171,384.366,388.230,174.761,36.311,156.824
C00704=1063.179,384.612,388.190,174.767,36.318,156.826
C00705=1063.186,384.859,388.150,174.772,36.325,156.828
C00706=1063.194,385.106,388.110,174.777,36.332,156.829
C00707=1063.200,385.352,388.069,174.782,36.339,156.831
C00708=1063.208,385.599,388.029,174.788,36.346,156.833
C00709=1063.216,385.845,387.988,174.793,36.353,156.834
C00710=1063.222,386.091,387.948,174.798,36.360,156.836
C00711=1063.230,386.338,387.908,174.804,36.367,156.838
C00712=1063.239,386.623,387.861,174.809,36.376,156.840
C00713=1063.248,386.907,387.814,174.815,36.384,156.842
C00714=1063.256,387.191,387.768,174.821,36.392,156.844
C00715=1063.265,387.476,387.721,174.827,36.400,156.846
C00716=1063.272,387.722,387.680,174.833,36.407,156.847
C00717=1063.280,387.969,387.640,174.838,36.414,156.849
C00718=1063.287,388.216,387.598,174.844,36.421,156.851
C00719=1063.295,388.462,387.558,174.849,36.429,156.853
C00720=1063.302,388.708,387.517,174.854,36.436,156.854
C00721=1063.310,388.955,387.477,174.860,36.443,156.856
C00722=1063.317,389.202,387.436,174.865,36.450,156.858
C00723=1063.325,389.448,387.395,174.870,36.458,156.860
C00724=1063.332,389.694,387.354,174.876,36.465,156.861
C00725=1063.340,389.941,387.313,174.881,36.472,156.863
C00726=1063.347,390.187,387.272,174.887,36.480,156.865
C00727=1063.355,390.434,387.231,174.892,36.487,156.867
C00728=1063.363,390.680,387.190,174.898,36.495,156.868
C00729=1063.370,390.927,387.149,174.904,36.502,156.870
C00730=1063.378,391.173,387.108,174.909,36.509,156.872
C00731=1063.385,391.420,387.067,174.915,36.517,156.874
C00732=1063.393,391.666,387.026,174.920,36.525,156.876
C00733=1063.401,391.913,386.985,174.926,36.532,156.877
C00734=1063.408,392.159,386.944,174.931,36.539,156.879
C00735=1063.416,392.405,386.902,174.937,36.547,156.881
C00736=1063.423,392.652,386.861,174.942,36.555,156.883
C00737=1063.431,392.898,386.820,174.948,36.562,156.885
C00738=1063.438,393.145,386.779,174.953,36.570,156.887
C00739=1063.446,393.391,386.737,174.960,36.577,156.889
C00740=1063.453,393.637,386.696,174.965,36.585,156.890
C00741=1063.461,393.883,386.654,174.970,36.593,156.892
C00742=1063.469,394.129,386.613,174.976,36.600,156.894
C00743=1063.476,394.376,386.572,174.981,36.608,156.896
C00744=1063.484,394.622,386.530,174.987,36.615,156.898
C00745=1063.491,394.869,386.489,174.993,36.623,156.900
C00746=1063.498,395.115,386.447,174.999,36.631,156.902
C00747=1063.506,395.362,386.405,175.005,36.639,156.904
C00748=1063.514,395.608,386.363,175.010,36.646,156.905
C00749=1063.521,395.854,386.321,175.016,36.654,156.907
C00750=1063.529,396.100,386.280,175.021,36.662,156.909
C00751=1063.536,396.346,386.238,175.027,36.670,156.911
C00752=1063.544,396.592,386.196,175.033,36.678,156.913
C00753=1063.552,396.840,386.155,175.039,36.686,156.915
C00754=1063.559,397.086,386.113,175.045,36.693,156.917
C00755=1063.568,397.331,386.071,175.050,36.702,156.919
C00756=1063.576,397.578,386.029,175.056,36.709,156.921
C00757=1063.583,397.825,385.987,175.062,36.717,156.923
C00758=1063.590,398.071,385.945,175.068,36.725,156.925
C00759=1063.598,398.317,385.903,175.074,36.733,156.927
C00760=1063.606,398.563,385.861,175.079,36.742,156.929
C00761=1063.613,398.809,385.819,175.086,36.750,156.931
C00762=1063.622,399.056,385.777,175.091,36.757,156.933
C00763=1063.629,399.302,385.735,175.097,36.765,156.935
C00764=1063.636,399.548,385.692,175.103,36.774,156.937
C00765=1063.644,399.795,385.650,175.109,36.782,156.939
C00766=1063.652,400.041,385.608,175.115,36.790,156.941
C00767=1063.660,400.288,385.566,175.121,36.798,156.943
C00768=1063.670,400.609,385.510,175.129,36.809,156.946
C00769=1063.681,400.931,385.455,175.137,36.820,156.948
C00770=1063.691,401.253,385.399,175.144,36.831,156.951
C00771=1063.701,401.575,385.344,175.152,36.841,156.954
C00772=1063.709,401.822,385.301,175.158,36.849,156.956
C00773=1063.716,402.068,385.259,175.165,36.858,156.958
C00774=1063.724,402.314,385.217,175.171,36.866,156.960
C00775=1063.733,402.560,385.174,175.176,36.875,156.962
C00776=1063.740,402.807,385.131,175.183,36.883,156.964
C00777=1063.748,403.053,385.088,175.189,36.891,156.966
C00778=1063.756,403.299,385.046,175.196,36.900,156.968
C00779=1063.764,403.545,385.002,175.201,36.908,156.970
C00780=1063.772,403.792,384.960,175.207,36.917,156.972
C00781=1063.779,404.037,384.917,175.214,36.925,156.975
C00782=1063.787,404.284,384.875,175.220,36.934,156.977
C00783=1063.796,404.530,384.831,175.227,36.942,156.979
C00784=1063.803,404.776,384.788,175.233,36.951,156.981
C00785=1063.811,405.022,384.745,175.238,36.959,156.983
C00786=1063.819,405.269,384.702,175.245,36.968,156.985
C00787=1063.827,405.514,384.660,175.251,36.977,156.987
C00788=1063.835,405.760,384.616,175.258,36.985,156.990
C00789=1063.843,406.006,384.573,175.264,36.994,156.992
C00790=1063.851,406.253,384.529,175.271,37.003,156.994
C00791=1063.858,406.499,384.486,175.277,37.011,156.996
C00792=1063.866,406.745,384.444,175.283,37.020,156.999
C00793=1063.874,406.992,384.400,175.289,37.029,157.001
C00794=1063.883,407.237,384.356,175.296,37.038,157.003
C00795=1063.891,407.483,384.313,175.302,37.047,157.005
C00796=1063.898,407.729,384.270,175.309,37.056,157.007
C00797=1063.906,407.975,384.227,175.315,37.065,157.010
C00798=1063.914,408.221,384.183,175.322,37.073,157.012
C00799=1063.922,408.468,384.139,175.328,37.082,157.014
C00800=1063.930,408.714,384.096,175.335,37.091,157.017
C00801=1063.938,408.960,384.052,175.341,37.101,157.019
C00802=1063.946,409.206,384.008,175.348,37.110,157.021
C00803=1063.955,409.452,383.965,175.354,37.119,157.023
C00804=1063.963,409.698,383.921,175.361,37.128,157.026
C00805=1063.970,409.944,383.877,175.367,37.137,157.028
C00806=1063.978,410.190,383.834,175.374,37.146,157.030
C00807=1063.987,410.436,383.790,175.381,37.155,157.033
C00808=1063.995,410.682,383.746,175.387,37.164,157.035
C00809=1064.003,410.928,383.702,175.394,37.173,157.037
C00810=1064.011,411.174,383.659,175.400,37.183,157.040
C00811=1064.019,411.420,383.615,175.408,37.192,157.042
C00812=1064.027,411.666,383.571,175.415,37.201,157.044
C00813=1064.035,411.912,383.527,175.421,37.210,157.047
C00814=1064.044,412.157,383.483,175.428,37.219,157.049
C00815=1064.052,412.404,383.439,175.435,37.229,157.052
C00816=1064.060,412.650,383.395,175.441,37.238,157.054
C00817=1064.068,412.896,383.350,175.448,37.247,157.056
C00818=1064.077,413.142,383.306,175.456,37.257,157.059
C00819=1064.085,413.387,383.262,175.462,37.266,157.061
C00820=1064.093,413.613,383.221,175.469,37.275,157.063
C00821=1064.101,413.838,383.181,175.474,37.283,157.066
C00822=1064.108,414.063,383.141,175.481,37.292,157.068
C00823=1064.116,414.288,383.100,175.488,37.301,157.070
C00824=1064.126,414.594,383.045,175.496,37.312,157.073
C00825=1064.136,414.900,382.990,175.505,37.325,157.076
C00826=1064.147,415.206,382.934,175.513,37.337,157.079
C00827=1064.157,415.512,382.879,175.522,37.348,157.082
C00828=1064.165,415.758,382.834,175.529,37.358,157.085
C00829=1064.173,416.003,382.789,175.537,37.368,157.087
C00830=1064.181,416.250,382.744,175.544,37.378,157.090
C00831=1064.190,416.495,382.700,175.551,37.387,157.093
C00832=1064.199,416.741,382.654,175.558,37.397,157.095
C00833=1064.207,416.987,382.610,175.565,37.407,157.098
C00834=1064.215,417.233,382.566,175.572,37.417,157.100
C00835=1064.224,417.479,382.520,175.580,37.427,157.103
C00836=1064.232,417.724,382.476,175.587,37.437,157.105
C00837=1064.241,417.970,382.430,175.594,37.447,157.108
C00838=1064.249,418.216,382.386,175.602,37.457,157.111
C00839=1064.257,418.462,382.340,175.609,37.467,157.113
C00840=1064.265,418.707,382.295,175.616,37.477,157.116
C00841=1064.274,418.954,382.250,175.623,37.487,157.119
C00842=1064.282,419.199,382.205,175.631,37.497,157.121
C00843=1064.291,419.444,382.160,175.638,37.507,157.124
C00844=1064.300,419.691,382.115,175.646,37.517,157.127
C00845=1064.308,419.936,382.070,175.653,37.527,157.129
C00846=1064.317,420.182,382.024,175.661,37.538,157.132
C00847=1064.326,420.428,381.979,175.668,37.548,157.135
C00848=1064.334,420.673,381.934,175.676,37.558,157.137
C00849=1064.342,420.919,381.888,175.683,37.568,157.140
C00850=1064.351,421.165,381.842,175.691,37.579,157.143
C00851=1064.360,421.410,381.797,175.698,37.589,157.145
C00852=1064.368,421.656,381.751,175.706,37.600,157.148
C00853=1064.377,421.902,381.706,175.713,37.610,157.151
C00854=1064.385,422.147,381.659,175.721,37.621,157.154
C00855=1064.394,422.393,381.614,175.729,37.631,157.156
C00856=1064.402,422.639,381.568,175.737,37.642,157.159
C00857=1064.411,422.885,381.523,175.745,37.652,157.162
C00858=1064.420,423.129,381.477,175.753,37.663,157.165
C00859=1064.428,423.375,381.431,175.760,37.674,157.168
C00860=1064.437,423.621,381.385,175.768,37.684,157.170
C00861=1064.445,423.867,381.339,175.776,37.695,157.173
C00862=1064.454,424.113,381.293,175.783,37.705,157.176
C00863=1064.463,424.358,381.246,175.792,37.716,157.179
C00864=1064.472,424.604,381.201,175.800,37.727,157.182
C00865=1064.480,424.849,381.154,175.808,37.738,157.185
C00866=1064.490,425.095,381.108,175.815,37.749,157.188
C00867=1064.497,425.340,381.063,175.823,37.760,157.191
C00868=1064.507,425.585,381.016,175.832,37.770,157.194
C00869=1064.515,425.831,380.970,175.840,37.781,157.196
C00870=1064.525,426.077,380.923,175.848,37.792,157.199
C00871=1064.534,426.322,380.876,175.855,37.803,157.202
C00872=1064.543,426.568,380.831,175.864,37.814,157.205
C00873=1064.551,426.814,380.784,175.872,37.825,157.208
C00874=1064.560,427.059,380.738,175.880,37.836,157.211
C00875=1064.569,427.304,380.691,175.888,37.847,157.214
C00876=1064.578,427.550,380.645,175.897,37.859,157.217
C00877=1064.586,427.795,380.598,175.905,37.870,157.220
C00878=1064.596,428.040,380.551,175.914,37.881,157.223
C00879=1064.604,428.285,380.504,175.922,37.892,157.226
C00880=1064.616,428.612,380.443,175.933,37.907,157.230
C00881=1064.627,428.938,380.380,175.943,37.923,157.235
C00882=1064.640,429.264,380.317,175.955,37.938,157.239
C00883=1064.652,429.589,380.255,175.966,37.953,157.243
C00884=1064.661,429.835,380.208,175.974,37.964,157.246
C00885=1064.670,430.080,380.160,175.984,37.976,157.249
C00886=1064.679,430.326,380.114,175.992,37.988,157.252
C00887=1064.688,430.571,380.066,176.001,37.999,157.255
C00888=1064.697,430.817,380.020,176.009,38.011,157.259
C00889=1064.706,431.062,379.972,176.018,38.022,157.262
C00890=1064.715,431.307,379.924,176.026,38.034,157.265
C00891=1064.724,431.553,379.878,176.035,38.046,157.268
C00892=1064.733,431.798,379.830,176.044,38.058,157.271
C00893=1064.742,432.043,379.782,176.052,38.070,157.275
C00894=1064.751,432.288,379.735,176.062,38.081,157.278
C00895=1064.760,432.534,379.687,176.070,38.093,157.281
C00896=1064.769,432.779,379.640,176.079,38.105,157.284
C00897=1064.779,433.024,379.592,176.088,38.118,157.288
C00898=1064.788,433.269,379.544,176.097,38.129,157.291
C00899=1064.797,433.515,379.497,176.106,38.141,157.294
C00900=1064.806,433.759,379.448,176.115,38.153,157.298
C00901=1064.816,434.004,379.401,176.124,38.166,157.301
C00902=1064.825,434.249,379.353,176.133,38.178,157.304
C00903=1064.834,434.495,379.305,176.142,38.190,157.308
C00904=1064.843,434.740,379.256,176.151,38.202,157.311
C00905=1064.852,434.985,379.209,176.161,38.215,157.314
C00906=1064.861,435.231,379.161,176.169,38.227,157.318
C00907=1064.871,435.476,379.112,176.179,38.239,157.321
C00908=1064.880,435.720,379.064,176.188,38.251,157.325
C00909=1064.890,435.966,379.017,176.197,38.264,157.328
C00910=1064.899,436.211,378.968,176.207,38.276,157.332
C00911=1064.909,436.456,378.920,176.216,38.289,157.335
C00912=1064.918,436.700,378.872,176.226,38.301,157.339
C00913=1064.927,436.946,378.823,176.234,38.314,157.342
C00914=1064.937,437.191,378.774,176.244,38.326,157.346
C00915=1064.946,437.436,378.727,176.253,38.339,157.349
C00916=1064.956,437.681,378.678,176.263,38.352,157.353
C00917=1064.966,437.926,378.629,176.273,38.365,157.356
C00918=1064.976,438.171,378.581,176.282,38.377,157.360
C00919=1064.985,438.416,378.532,176.292,38.390,157.363
C00920=1064.994,438.661,378.483,176.301,38.403,157.367
C00921=1065.004,438.906,378.433,176.312,38.416,157.371
C00922=1065.013,439.151,378.385,176.322,38.429,157.374
C00923=1065.023,439.396,378.336,176.331,38.442,157.378
C00924=1065.032,439.641,378.287,176.341,38.455,157.382
C00925=1065.042,439.886,378.238,176.351,38.468,157.385
C00926=1065.052,440.131,378.190,176.360,38.481,157.389
C00927=1065.061,440.376,378.140,176.370,38.494,157.393
C00928=1065.071,440.620,378.091,176.381,38.508,157.397
C00929=1065.080,440.865,378.041,176.391,38.521,157.400
C00930=1065.090,441.110,377.993,176.401,38.534,157.404
C00931=1065.100,441.355,377.943,176.410,38.548,157.408
C00932=1065.110,441.600,377.893,176.421,38.561,157.412
C00933=1065.119,441.845,377.844,176.431,38.574,157.416
C00934=1065.129,442.089,377.795,176.441,38.588,157.419
C00935=1065.139,442.335,377.745,176.452,38.602,157.423
C00936=1065.156,442.743,377.662,176.468,38.624,157.430
C00937=1065.172,443.152,377.579,176.486,38.647,157.436
C00938=1065.189,443.560,377.496,176.504,38.670,157.443
C00939=1065.205,443.969,377.413,176.522,38.693,157.449
C00940=1065.215,444.214,377.363,176.532,38.707,157.453
C00941=1065.225,444.458,377.313,176.543,38.721,157.457
C00942=1065.235,444.703,377.263,176.553,38.735,157.461
C00943=1065.244,444.948,377.213,176.564,38.749,157.466
C00944=1065.255,445.192,377.163,176.574,38.763,157.470
C00945=1065.265,445.437,377.113,176.585,38.777,157.474
C00946=1065.275,445.682,377.062,176.596,38.791,157.478
C00947=1065.284,445.926,377.011,176.607,38.805,157.482
C00948=1065.295,446.171,376.962,176.618,38.820,157.486
C00949=1065.305,446.415,376.911,176.629,38.834,157.490
C00950=1065.315,446.660,376.860,176.639,38.848,157.494
C00951=1065.326,446.904,376.810,176.651,38.862,157.498
C00952=1065.336,447.148,376.759,176.662,38.877,157.503
C00953=1065.346,447.392,376.709,176.673,38.891,157.507
C00954=1065.356,447.637,376.658,176.685,38.906,157.511
C00955=1065.367,447.881,376.608,176.695,38.920,157.515
C00956=1065.378,448.124,376.559,176.707,38.934,157.519
C00957=1065.391,448.368,376.510,176.718,38.948,157.524
C00958=1065.404,448.612,376.461,176.729,38.961,157.527
C00959=1065.420,448.858,376.414,176.741,38.975,157.531
C00960=1065.435,449.103,376.367,176.753,38.988,157.535
C00961=1065.452,449.347,376.320,176.764,39.000,157.539
C00962=1065.470,449.593,376.275,176.775,39.012,157.543
C00963=1065.488,449.838,376.230,176.786,39.024,157.546
C00964=1065.149,449.843,375.964,176.777,39.149,157.580
C00965=1065.130,449.598,376.009,176.766,39.138,157.577
C00966=1065.112,449.353,376.054,176.755,39.126,157.573
C00967=1065.095,449.107,376.101,176.743,39.113,157.569
C00968=1065.079,448.863,376.147,176.732,39.100,157.565
C00969=1065.064,448.617,376.195,176.720,39.087,157.561
C00970=1065.050,448.373,376.244,176.709,39.074,157.558
C00971=1065.037,448.130,376.293,176.697,39.060,157.553
C00972=1065.026,447.886,376.342,176.685,39.046,157.549
C00973=1065.015,447.642,376.392,176.674,39.032,157.545
C00974=1065.004,447.397,376.443,176.663,39.018,157.541
C00975=1064.995,447.153,376.493,176.651,39.003,157.537
C00976=1064.984,446.910,376.544,176.641,38.989,157.532
C00977=1064.974,446.666,376.595,176.629,38.974,157.528
C00978=1064.964,446.420,376.645,176.618,38.960,157.524
C00979=1064.954,446.176,376.696,176.607,38.946,157.520
C00980=1064.943,445.932,376.746,176.596,38.932,157.516
C00981=1064.933,445.687,376.797,176.585,38.918,157.512
C00982=1064.924,445.442,376.847,176.574,38.904,157.508
C00983=1064.913,445.198,376.897,176.563,38.890,157.503
C00984=1064.903,444.953,376.947,176.553,38.876,157.499
C00985=1064.893,444.709,376.998,176.542,38.862,157.495
C00986=1064.883,444.463,377.048,176.531,38.848,157.491
C00987=1064.873,444.219,377.098,176.520,38.834,157.487
C00988=1064.863,443.975,377.148,176.509,38.820,157.483
C00989=1064.848,443.585,377.227,176.492,38.798,157.477
C00990=1064.831,443.196,377.307,176.476,38.776,157.471
C00991=1064.815,442.806,377.386,176.459,38.754,157.464
C00992=1064.800,442.417,377.465,176.443,38.733,157.458
C00993=1064.790,442.172,377.515,176.432,38.719,157.454
C00994=1064.780,441.927,377.564,176.422,38.706,157.450
C00995=1064.770,441.682,377.613,176.411,38.692,157.447
C00996=1064.761,441.438,377.663,176.401,38.679,157.443
C00997=1064.750,441.193,377.713,176.391,38.666,157.439
C00998=1064.741,440.947,377.762,176.380,38.652,157.435
C00999=1064.731,440.703,377.811,176.371,38.639,157.431
C01000=1064.722,440.458,377.861,176.361,38.626,157.428
C01001=1064.712,440.213,377.909,176.351,38.613,157.424
C01002=1064.702,439.968,377.960,176.340,38.600,157.420
C01003=1064.693,439.723,378.008,176.331,38.587,157.416
C01004=1064.683,439.478,378.057,176.321,38.574,157.413
C01005=1064.673,439.233,378.106,176.311,38.561,157.409
C01006=1064.664,438.988,378.155,176.302,38.548,157.405
C01007=1064.655,438.743,378.204,176.291,38.535,157.402
C01008=1064.645,438.499,378.253,176.281,38.522,157.398
C01009=1064.635,438.254,378.302,176.272,38.509,157.395
C01010=1064.626,438.008,378.351,176.262,38.497,157.391
C01011=1064.616,437.763,378.399,176.252,38.484,157.387
C01012=1064.606,437.519,378.448,176.243,38.471,157.384
C01013=1064.597,437.274,378.497,176.233,38.458,157.380
C01014=1064.587,437.028,378.544,176.224,38.446,157.377
C01015=1064.577,436.783,378.593,176.214,38.434,157.373
C01016=1064.568,436.539,378.641,176.205,38.421,157.370
C01017=1064.559,436.293,378.690,176.195,38.409,157.366
C01018=1064.550,436.048,378.738,176.186,38.396,157.363
C01019=1064.540,435.803,378.787,176.176,38.383,157.359
C01020=1064.530,435.558,378.835,176.167,38.371,157.356
C01021=1064.521,435.313,378.882,176.157,38.359,157.352
C01022=1064.512,435.068,378.931,176.149,38.347,157.349
C01023=1064.502,434.822,378.979,176.140,38.334,157.346
C01024=1064.493,434.578,379.027,176.130,38.322,157.342
C01025=1064.484,434.333,379.075,176.121,38.310,157.339
C01026=1064.474,434.087,379.123,176.111,38.298,157.335
C01027=1064.466,433.842,379.171,176.102,38.286,157.332
C01028=1064.456,433.597,379.219,176.094,38.273,157.329
C01029=1064.447,433.351,379.267,176.085,38.262,157.325
C01030=1064.438,433.106,379.314,176.075,38.250,157.322
C01031=1064.428,432.861,379.362,176.066,38.237,157.319
C01032=1064.419,432.616,379.410,176.058,38.226,157.315
C01033=1064.410,432.371,379.458,176.049,38.214,157.312
C01034=1064.401,432.126,379.506,176.039,38.202,157.309
C01035=1064.392,431.881,379.553,176.031,38.190,157.306
C01036=1064.383,431.635,379.600,176.022,38.178,157.302
C01037=1064.374,431.390,379.648,176.013,38.166,157.299
C01038=1064.365,431.144,379.695,176.005,38.155,157.296
C01039=1064.356,430.899,379.743,175.996,38.143,157.293
C01040=1064.346,430.654,379.791,175.986,38.131,157.289
C01041=1064.338,430.408,379.837,175.978,38.120,157.286
C01042=1064.328,430.164,379.884,175.969,38.108,157.283
C01043=1064.319,429.918,379.931,175.961,38.097,157.280
C01044=1064.310,429.673,379.979,175.952,38.086,157.277
C01045=1064.298,429.345,380.042,175.941,38.070,157.273
C01046=1064.286,429.017,380.105,175.930,38.055,157.269
C01047=1064.274,428.689,380.168,175.918,38.040,157.264
C01048=1064.263,428.361,380.229,175.907,38.025,157.260
C01049=1064.253,428.117,380.276,175.899,38.014,157.257
C01050=1064.244,427.871,380.323,175.890,38.002,157.254
C01051=1064.236,427.626,380.370,175.882,37.991,157.251
C01052=1064.227,427.379,380.417,175.873,37.980,157.248
C01053=1064.217,427.134,380.463,175.865,37.969,157.245
C01054=1064.209,426.889,380.510,175.858,37.958,157.242
C01055=1064.200,426.643,380.556,175.849,37.947,157.239
C01056=1064.191,426.398,380.603,175.841,37.935,157.236
C01057=1064.183,426.152,380.649,175.832,37.924,157.233
C01058=1064.173,425.907,380.695,175.824,37.914,157.230
C01059=1064.165,425.662,380.742,175.816,37.903,157.227
C01060=1064.155,425.416,380.788,175.808,37.892,157.224
C01061=1064.147,425.170,380.834,175.800,37.881,157.221
C01062=1064.138,424.925,380.880,175.792,37.870,157.219
C01063=1064.129,424.680,380.927,175.784,37.859,157.216
C01064=1064.120,424.434,380.973,175.776,37.849,157.213
C01065=1064.112,424.188,381.019,175.768,37.838,157.210
C01066=1064.103,423.943,381.066,175.760,37.827,157.207
C01067=1064.094,423.697,381.112,175.752,37.817,157.204
C01068=1064.085,423.452,381.158,175.744,37.806,157.201
C01069=1064.076,423.206,381.203,175.737,37.795,157.199
C01070=1064.068,422.960,381.249,175.728,37.785,157.196
C01071=1064.059,422.715,381.295,175.720,37.775,157.193
C01072=1064.051,422.469,381.341,175.713,37.764,157.190
C01073=1064.042,422.223,381.386,175.705,37.753,157.187
C01074=1064.033,421.978,381.433,175.698,37.743,157.185
C01075=1064.025,421.733,381.478,175.690,37.732,157.182
C01076=1064.017,421.487,381.524,175.682,37.722,157.179
C01077=1064.008,421.241,381.569,175.675,37.712,157.176
C01078=1063.999,420.995,381.615,175.666,37.701,157.174
C01079=1063.991,420.749,381.661,175.659,37.691,157.171
C01080=1063.982,420.504,381.706,175.651,37.681,157.168
C01081=1063.973,420.258,381.751,175.644,37.670,157.165
C01082=1063.965,420.013,381.796,175.636,37.660,157.163
C01083=1063.957,419.767,381.842,175.629,37.650,157.160
C01084=1063.948,419.521,381.888,175.621,37.640,157.157
C01085=1063.939,419.276,381.933,175.614,37.630,157.155
C01086=1063.931,419.029,381.978,175.606,37.620,157.152
C01087=1063.922,418.784,382.023,175.599,37.610,157.149
C01088=1063.913,418.538,382.068,175.591,37.600,157.147
C01089=1063.904,418.292,382.114,175.584,37.590,157.144
C01090=1063.897,418.046,382.158,175.576,37.580,157.142
C01091=1063.888,417.800,382.204,175.570,37.570,157.139
C01092=1063.880,417.555,382.248,175.562,37.560,157.136
C01093=1063.871,417.309,382.294,175.555,37.550,157.134
C01094=1063.863,417.063,382.338,175.548,37.540,157.131
C01095=1063.854,416.818,382.383,175.540,37.531,157.129
C01096=1063.846,416.572,382.428,175.533,37.521,157.126
C01097=1063.837,416.326,382.473,175.526,37.511,157.124
C01098=1063.829,416.080,382.517,175.518,37.501,157.121
C01099=1063.821,415.834,382.562,175.511,37.492,157.118
C01100=1063.813,415.588,382.607,175.505,37.482,157.116
C01101=1063.802,415.281,382.663,175.495,37.469,157.113
C01102=1063.792,414.973,382.719,175.487,37.457,157.110
C01103=1063.782,414.664,382.774,175.478,37.446,157.106
C01104=1063.772,414.357,382.830,175.468,37.434,157.103
C01105=1063.763,414.111,382.875,175.462,37.424,157.101
C01106=1063.754,413.865,382.919,175.455,37.414,157.098
C01107=1063.746,413.619,382.963,175.448,37.405,157.096
C01108=1063.738,413.373,383.008,175.441,37.396,157.094
C01109=1063.730,413.127,383.052,175.434,37.386,157.091
C01110=1063.722,412.881,383.096,175.427,37.377,157.089
C01111=1063.712,412.635,383.140,175.420,37.368,157.086
C01112=1063.704,412.389,383.184,175.413,37.358,157.084
C01113=1063.696,412.143,383.228,175.407,37.349,157.082
C01114=1063.688,411.898,383.273,175.399,37.340,157.079
C01115=1063.680,411.651,383.316,175.392,37.331,157.077
C01116=1063.672,411.406,383.360,175.386,37.321,157.074
C01117=1063.663,411.159,383.405,175.379,37.312,157.072
C01118=1063.655,410.913,383.448,175.372,37.303,157.070
C01119=1063.646,410.667,383.492,175.366,37.294,157.067
C01120=1063.639,410.421,383.536,175.359,37.285,157.065
C01121=1063.631,410.175,383.580,175.352,37.276,157.063
C01122=1063.622,409.929,383.623,175.346,37.267,157.060
C01123=1063.614,409.684,383.667,175.339,37.257,157.058
C01124=1063.606,409.437,383.711,175.333,37.248,157.056
C01125=1063.598,409.191,383.754,175.326,37.239,157.053
C01126=1063.590,408.945,383.798,175.319,37.230,157.051
C01127=1063.582,408.699,383.842,175.313,37.222,157.049
C01128=1063.574,408.453,383.886,175.306,37.213,157.047
C01129=1063.565,408.207,383.929,175.300,37.204,157.044
C01130=1063.558,407.962,383.973,175.293,37.195,157.042
C01131=1063.550,407.715,384.016,175.287,37.186,157.040
C01132=1063.542,407.469,384.059,175.280,37.177,157.037
C01133=1063.534,407.223,384.103,175.273,37.168,157.035
C01134=1063.526,406.977,384.146,175.267,37.159,157.033
C01135=1063.518,406.730,384.190,175.260,37.151,157.031
C01136=1063.511,406.485,384.233,175.254,37.142,157.028
C01137=1063.502,406.239,384.276,175.247,37.133,157.026
C01138=1063.494,405.992,384.319,175.241,37.124,157.024
C01139=1063.487,405.746,384.363,175.235,37.116,157.022
C01140=1063.478,405.500,384.406,175.229,37.107,157.020
C01141=1063.470,405.255,384.449,175.222,37.098,157.018
C01142=1063.463,405.008,384.492,175.216,37.090,157.015
C01143=1063.454,404.761,384.535,175.209,37.081,157.013
C01144=1063.447,404.515,384.578,175.203,37.073,157.011
C01145=1063.439,404.270,384.621,175.196,37.064,157.009
C01146=1063.431,404.023,384.664,175.191,37.056,157.007
C01147=1063.423,403.777,384.707,175.185,37.047,157.005
C01148=1063.415,403.531,384.750,175.178,37.038,157.002
C01149=1063.407,403.284,384.793,175.172,37.030,157.000
C01150=1063.399,403.039,384.835,175.166,37.022,156.998
C01151=1063.392,402.792,384.878,175.160,37.013,156.996
C01152=1063.384,402.546,384.921,175.154,37.005,156.994
C01153=1063.374,402.250,384.972,175.146,36.995,156.991
C01154=1063.364,401.953,385.023,175.139,36.985,156.989
C01155=1063.355,401.656,385.074,175.132,36.975,156.986
C01156=1063.345,401.360,385.126,175.124,36.965,156.984
C01157=1063.337,401.107,385.170,175.118,36.957,156.982
C01158=1063.330,400.855,385.213,175.111,36.948,156.980
C01159=1063.321,400.602,385.256,175.106,36.940,156.978
C01160=1063.314,400.349,385.300,175.099,36.932,156.976
C01161=1063.306,400.104,385.342,175.093,36.923,156.974
C01162=1063.298,399.857,385.385,175.087,36.915,156.972
C01163=1063.290,399.611,385.427,175.081,36.907,156.970
C01164=1063.282,399.365,385.469,175.075,36.899,156.968
C01165=1063.275,399.119,385.511,175.069,36.891,156.966
C01166=1063.267,398.873,385.553,175.064,36.883,156.964
C01167=1063.259,398.626,385.596,175.057,36.875,156.962
C01168=1063.251,398.380,385.638,175.052,36.867,156.960
C01169=1063.244,398.134,385.680,175.046,36.859,156.957
C01170=1063.236,397.887,385.722,175.039,36.851,156.956
C01171=1063.229,397.641,385.764,175.034,36.843,156.954
C01172=1063.221,397.395,385.806,175.028,36.835,156.952
C01173=1063.213,397.148,385.848,175.023,36.827,156.950
C01174=1063.205,396.902,385.889,175.016,36.819,156.948
C01175=1063.197,396.656,385.931,175.010,36.811,156.946
C01176=1063.189,396.409,385.973,175.005,36.804,156.944
C01177=1063.182,396.163,386.015,174.999,36.796,156.942
C01178=1063.174,395.917,386.057,174.993,36.788,156.940
C01179=1063.167,395.671,386.099,174.987,36.780,156.938
C01180=1063.159,395.424,386.140,174.982,36.772,156.936
C01181=1063.151,395.178,386.182,174.976,36.765,156.934
C01182=1063.144,394.931,386.223,174.970,36.757,156.932
C01183=1063.136,394.685,386.265,174.964,36.750,156.931
C01184=1063.129,394.439,386.307,174.958,36.741,156.929
C01185=1063.122,394.192,386.349,174.953,36.734,156.927
C01186=1063.114,393.946,386.390,174.947,36.726,156.925
C01187=1063.106,393.700,386.431,174.942,36.719,156.923
C01188=1063.099,393.454,386.472,174.936,36.711,156.921
C01189=1063.090,393.207,386.515,174.930,36.703,156.919
C01190=1063.083,392.960,386.556,174.924,36.696,156.917
C01191=1063.076,392.714,386.597,174.919,36.688,156.915
C01192=1063.068,392.468,386.638,174.913,36.681,156.914
C01193=1063.060,392.221,386.680,174.908,36.674,156.912
C01194=1063.053,391.975,386.721,174.903,36.666,156.910
C01195=1063.045,391.729,386.762,174.897,36.658,156.908
C01196=1063.037,391.483,386.803,174.891,36.651,156.906
C01197=1063.030,391.236,386.845,174.885,36.644,156.905
C01198=1063.023,390.989,386.886,174.880,36.636,156.903
C01199=1063.015,390.743,386.927,174.874,36.628,156.901
C01200=1063.008,390.497,386.967,174.869,36.621,156.899
C01201=1063.001,390.251,387.009,174.864,36.614,156.897
C01202=1062.993,390.004,387.049,174.858,36.607,156.896
C01203=1062.985,389.758,387.091,174.853,36.599,156.894
C01204=1062.977,389.512,387.131,174.847,36.592,156.892
C01205=1062.970,389.265,387.172,174.842,36.585,156.890
C01206=1062.962,389.018,387.212,174.837,36.578,156.889
C01207=1062.955,388.771,387.254,174.830,36.570,156.887
C01208=1062.947,388.525,387.294,174.825,36.563,156.885
C01209=1062.939,388.279,387.335,174.819,36.556,156.883
C01210=1062.932,388.032,387.376,174.814,36.549,156.882
C01211=1062.924,387.785,387.416,174.809,36.542,156.880
C01212=1062.917,387.539,387.457,174.803,36.535,156.878
C01213=1062.908,387.253,387.504,174.797,36.526,156.876
C01214=1062.900,386.967,387.552,174.791,36.518,156.874
C01215=1062.891,386.680,387.598,174.785,36.509,156.872
C01216=1062.883,386.394,387.645,174.778,36.501,156.870
C01217=1062.875,386.148,387.686,174.773,36.494,156.868
C01218=1062.868,385.901,387.726,174.768,36.487,156.867
C01219=1062.860,385.655,387.767,174.762,36.480,156.865
C01220=1062.852,385.408,387.807,174.757,36.473,156.863
C01221=1062.845,385.162,387.848,174.752,36.466,156.862
C01222=1062.838,384.916,387.887,174.747,36.459,156.860
C01223=1062.831,384.668,387.928,174.742,36.452,156.858
C01224=1062.823,384.422,387.969,174.737,36.445,156.857
C01225=1062.816,384.176,388.008,174.732,36.438,156.855
C01226=1062.809,383.929,388.049,174.727,36.432,156.853
C01227=1062.801,383.682,388.089,174.721,36.424,156.852
C01228=1062.794,383.436,388.129,174.716,36.417,156.850
C01229=1062.787,383.189,388.169,174.711,36.411,156.848
C01230=1062.779,382.943,388.210,174.706,36.404,156.847
C01231=1062.772,382.696,388.250,174.700,36.397,156.845
C01232=1062.765,382.449,388.290,174.695,36.390,156.843
C01233=1062.758,382.203,388.330,174.690,36.383,156.842
C01234=1062.751,381.956,388.370,174.685,36.376,156.840
C01235=1062.743,381.710,388.410,174.680,36.369,156.839
C01236=1062.736,381.463,388.450,174.675,36.363,156.837
C01237=1062.729,381.216,388.490,174.669,36.356,156.835
C01238=1062.721,380.970,388.530,174.664,36.349,156.834
C01239=1062.715,380.723,388.569,174.659,36.343,156.832
C01240=1062.707,380.476,388.609,174.654,36.336,156.831
C01241=1062.700,380.230,388.649,174.650,36.329,156.829
C01242=1062.692,379.983,388.689,174.645,36.322,156.827
C01243=1062.685,379.737,388.728,174.639,36.316,156.826
C01244=1062.677,379.490,388.768,174.634,36.309,156.824
C01245=1062.670,379.244,388.808,174.629,36.302,156.823
C01246=1062.663,378.996,388.847,174.624,36.296,156.821
C01247=1062.656,378.750,388.887,174.619,36.290,156.820
C01248=1062.648,378.503,388.927,174.614,36.283,156.818
C01249=1062.641,378.257,388.966,174.609,36.276,156.816
C01250=1062.634,378.009,389.006,174.604,36.270,156.815
C01251=1062.627,377.763,389.045,174.599,36.263,156.813
C01252=1062.620,377.517,389.085,174.594,36.256,156.812
C01253=1062.612,377.269,389.124,174.589,36.250,156.810
C01254=1062.605,377.023,389.164,174.584,36.244,156.809
C01255=1062.598,376.776,389.202,174.579,36.237,156.807
C01256=1062.591,376.529,389.242,174.574,36.230,156.806
C01257=1062.584,376.282,389.281,174.570,36.224,156.804
C01258=1062.577,376.036,389.321,174.565,36.218,156.803
C01259=1062.569,375.789,389.360,174.560,36.211,156.801
C01260=1062.562,375.542,389.399,174.555,36.205,156.800
C01261=1062.555,375.296,389.438,174.550,36.198,156.798
C01262=1062.547,375.049,389.478,174.545,36.192,156.797
C01263=1062.540,374.802,389.516,174.541,36.186,156.795
C01264=1062.533,374.555,389.555,174.536,36.180,156.794
C01265=1062.526,374.309,389.595,174.531,36.173,156.792
C01266=1062.519,374.062,389.634,174.526,36.167,156.791
C01267=1062.512,373.815,389.673,174.521,36.160,156.789
C01268=1062.505,373.568,389.712,174.517,36.154,156.788
C01269=1062.498,373.313,389.752,174.511,36.147,156.786
C01270=1062.491,373.057,389.793,174.506,36.141,156.785
C01271=1062.483,372.802,389.833,174.501,36.135,156.783
C01272=1062.476,372.547,389.874,174.496,36.128,156.782
C01273=1062.469,372.300,389.912,174.491,36.122,156.780
C01274=1062.462,372.053,389.951,174.487,36.115,156.779
C01275=1062.454,371.806,389.990,174.482,36.109,156.777
C01276=1062.447,371.559,390.029,174.477,36.103,156.776
C01277=1062.440,371.312,390.068,174.472,36.097,156.774
C01278=1062.433,371.066,390.106,174.468,36.091,156.773
C01279=1062.426,370.819,390.145,174.463,36.085,156.771
C01280=1062.419,370.572,390.183,174.458,36.078,156.770
C01281=1062.412,370.325,390.221,174.453,36.072,156.769
C01282=1062.404,370.077,390.260,174.449,36.066,156.767
C01283=1062.398,369.830,390.299,174.445,36.060,156.766
C01284=1062.390,369.584,390.337,174.440,36.054,156.764
C01285=1062.383,369.337,390.376,174.435,36.048,156.763
C01286=1062.376,369.091,390.414,174.431,36.042,156.762
C01287=1062.369,368.843,390.452,174.426,36.036,156.760
C01288=1062.362,368.596,390.491,174.421,36.030,156.759
C01289=1062.355,368.350,390.530,174.416,36.024,156.757
C01290=1062.348,368.102,390.568,174.412,36.018,156.756
C01291=1062.341,367.856,390.606,174.407,36.012,156.755
C01292=1062.334,367.609,390.645,174.402,36.006,156.753
C01293=1062.327,367.362,390.683,174.398,36.000,156.752
C01294=1062.320,367.115,390.721,174.394,35.994,156.750
C01295=1062.313,366.868,390.760,174.389,35.988,156.749
C01296=1062.306,366.621,390.797,174.384,35.982,156.748
C01297=1062.299,366.374,390.836,174.380,35.976,156.746
C01298=1062.292,366.127,390.874,174.375,35.970,156.745
C01299=1062.285,365.880,390.913,174.370,35.964,156.744
C01300=1062.278,365.633,390.951,174.367,35.958,156.742
C01301=1062.271,365.386,390.989,174.362,35.952,156.741
C01302=1062.265,365.140,391.027,174.357,35.947,156.740
C01303=1062.258,364.893,391.064,174.352,35.941,156.738
C01304=1062.251,364.646,391.103,174.348,35.935,156.737
C01305=1062.244,364.399,391.141,174.343,35.929,156.736
C01306=1062.237,364.152,391.180,174.339,35.923,156.734
C01307=1062.230,363.905,391.217,174.335,35.917,156.733
C01308=1062.223,363.657,391.255,174.330,35.911,156.732
C01309=1062.216,363.410,391.293,174.325,35.906,156.730
C01310=1062.209,363.164,391.330,174.321,35.900,156.729
C01311=1062.202,362.917,391.369,174.317,35.894,156.728
C01312=1062.195,362.670,391.406,174.312,35.888,156.726
C01313=1062.188,362.422,391.444,174.308,35.883,156.725
C01314=1062.181,362.175,391.482,174.303,35.877,156.724
C01315=1062.174,361.928,391.519,174.298,35.871,156.722
C01316=1062.168,361.681,391.557,174.295,35.865,156.721
C01317=1062.160,361.434,391.594,174.290,35.860,156.720
C01318=1062.154,361.187,391.632,174.285,35.854,156.718
C01319=1062.147,360.940,391.670,174.281,35.849,156.717
C01320=1062.140,360.693,391.707,174.277,35.843,156.716
C01321=1062.133,360.452,391.744,174.273,35.837,156.715
C01322=1062.126,360.209,391.781,174.268,35.832,156.713
C01323=1062.119,359.967,391.818,174.264,35.826,156.712
C01324=1062.112,359.725,391.854,174.260,35.820,156.711
C01325=1062.106,359.482,391.891,174.255,35.815,156.710
C01326=1062.099,359.240,391.928,174.251,35.810,156.708
C01327=1062.092,358.998,391.964,174.247,35.804,156.707
C01328=1062.086,358.755,392.001,174.242,35.798,156.706
C01329=1062.079,358.509,392.038,174.239,35.793,156.705
C01330=1062.072,358.261,392.076,174.234,35.788,156.703
C01331=1062.065,358.014,392.113,174.229,35.782,156.702
C01332=1062.058,357.767,392.150,174.226,35.777,156.701
C01333=1062.051,357.520,392.187,174.221,35.771,156.700
C01334=1062.044,357.273,392.225,174.217,35.765,156.698
C01335=1062.037,357.026,392.261,174.212,35.760,156.697
C01336=1062.030,356.779,392.299,174.208,35.755,156.696
C01337=1062.023,356.532,392.336,174.204,35.749,156.695
C01338=1062.017,356.285,392.373,174.199,35.744,156.693
C01339=1062.009,356.037,392.410,174.196,35.738,156.692
C01340=1062.003,355.790,392.447,174.191,35.732,156.691
C01341=1061.996,355.543,392.484,174.186,35.727,156.690
C01342=1061.990,355.295,392.522,174.183,35.722,156.688
C01343=1061.983,355.049,392.559,174.178,35.716,156.687
C01344=1061.976,354.801,392.596,174.175,35.711,156.686
C01345=1061.969,354.555,392.633,174.170,35.705,156.685
C01346=1061.962,354.307,392.669,174.166,35.700,156.684
C01347=1061.955,354.060,392.706,174.162,35.695,156.682
C01348=1061.948,353.813,392.743,174.157,35.690,156.681
C01349=1061.942,353.566,392.780,174.153,35.684,156.680
C01350=1061.935,353.318,392.816,174.149,35.679,156.679
C01351=1061.928,353.072,392.854,174.145,35.673,156.678
C01352=1061.921,352.824,392.890,174.141,35.668,156.676
C01353=1061.915,352.577,392.927,174.137,35.662,156.675
C01354=1061.908,352.330,392.964,174.132,35.657,156.674
C01355=1061.901,352.083,393.001,174.128,35.652,156.673
C01356=1061.894,351.835,393.038,174.124,35.646,156.672
C01357=1061.888,351.588,393.074,174.120,35.641,156.670
C01358=1061.881,351.340,393.111,174.116,35.636,156.669
C01359=1061.874,351.093,393.147,174.111,35.631,156.668
C01360=1061.867,350.847,393.184,174.108,35.625,156.667
C01361=1061.860,350.599,393.221,174.103,35.620,156.666
C01362=1061.854,350.352,393.257,174.100,35.615,156.664
C01363=1061.846,350.105,393.293,174.095,35.610,156.663
C01364=1061.840,349.858,393.330,174.092,35.604,156.662
C01365=1061.833,349.610,393.367,174.087,35.599,156.661
C01366=1061.827,349.363,393.403,174.082,35.594,156.660
C01367=1061.820,349.116,393.439,174.079,35.589,156.659
C01368=1061.813,348.868,393.476,174.074,35.584,156.658
C01369=1061.806,348.621,393.512,174.071,35.578,156.656
C01370=1061.800,348.374,393.548,174.066,35.573,156.655
C01371=1061.793,348.126,393.584,174.063,35.568,156.654
C01372=1061.786,347.879,393.621,174.058,35.563,156.653
C01373=1061.780,347.632,393.657,174.055,35.558,156.652
C01374=1061.772,347.385,393.693,174.050,35.553,156.651
C01375=1061.766,347.138,393.730,174.047,35.548,156.650
C01376=1061.760,346.890,393.765,174.042,35.542,156.648
C01377=1061.753,346.650,393.801,174.039,35.537,156.647
C01378=1061.747,346.410,393.835,174.034,35.533,156.646
C01379=1061.740,346.170,393.871,174.031,35.528,156.645
C01380=1061.733,345.930,393.906,174.027,35.523,156.644
C01381=1061.727,345.690,393.941,174.023,35.518,156.643
C01382=1061.721,345.450,393.976,174.019,35.513,156.642
C01383=1061.714,345.209,394.011,174.015,35.508,156.641
C01384=1061.707,344.970,394.046,174.011,35.503,156.640
C01385=1061.701,344.722,394.081,174.008,35.498,156.639
C01386=1061.694,344.474,394.118,174.003,35.493,156.637
C01387=1061.688,344.227,394.153,174.000,35.488,156.636
C01388=1061.681,343.980,394.190,173.995,35.483,156.635
C01389=1061.674,343.733,394.225,173.992,35.477,156.634
C01390=1061.668,343.486,394.261,173.987,35.473,156.633
C01391=1061.661,343.238,394.297,173.984,35.468,156.632
C01392=1061.654,342.990,394.333,173.979,35.463,156.631
C01393=1061.648,342.743,394.369,173.976,35.457,156.630
C01394=1061.641,342.496,394.404,173.972,35.453,156.629
C01395=1061.635,342.249,394.440,173.968,35.448,156.628
C01396=1061.628,342.001,394.475,173.965,35.443,156.627
C01397=1061.621,341.754,394.512,173.960,35.438,156.625
C01398=1061.614,341.506,394.547,173.957,35.433,156.624
C01399=1061.607,341.259,394.582,173.952,35.428,156.623
C01400=1061.601,341.012,394.619,173.949,35.423,156.622
C01401=1061.594,340.764,394.654,173.945,35.419,156.621
C01402=1061.587,340.517,394.689,173.941,35.413,156.620
C01403=1061.581,340.269,394.725,173.937,35.408,156.619
C01404=1061.574,340.023,394.761,173.933,35.404,156.618
C01405=1061.568,339.775,394.796,173.929,35.398,156.617
C01406=1061.561,339.527,394.832,173.926,35.394,156.616
C01407=1061.554,339.280,394.867,173.921,35.389,156.615
C01408=1061.547,339.032,394.902,173.918,35.384,156.614
C01409=1061.541,338.784,394.938,173.915,35.379,156.613
C01410=1061.535,338.537,394.973,173.910,35.374,156.612
C01411=1061.528,338.290,395.009,173.907,35.369,156.610
C01412=1061.521,338.043,395.045,173.902,35.365,156.609
C01413=1061.515,337.795,395.080,173.899,35.359,156.608
C01414=1061.508,337.548,395.115,173.895,35.355,156.607
C01415=1061.501,337.301,395.150,173.891,35.350,156.606
C01416=1061.495,337.053,395.186,173.887,35.345,156.605
C01417=1061.488,336.806,395.221,173.884,35.341,156.604
C01418=1061.482,336.558,395.256,173.880,35.336,156.603
C01419=1061.475,336.310,395.290,173.876,35.331,156.602
C01420=1061.468,336.063,395.325,173.873,35.326,156.601
C01421=1061.462,335.815,395.361,173.868,35.322,156.600
C01422=1061.455,335.568,395.396,173.865,35.316,156.599
C01423=1061.449,335.320,395.431,173.861,35.312,156.598
C01424=1061.443,335.074,395.466,173.857,35.307,156.597
C01425=1061.436,334.826,395.501,173.854,35.303,156.596
C01426=1061.429,334.578,395.536,173.850,35.298,156.595
C01427=1061.423,334.331,395.571,173.846,35.293,156.594
C01428=1061.416,334.084,395.606,173.842,35.288,156.593
C01429=1061.409,333.836,395.641,173.839,35.284,156.592
C01430=1061.403,333.588,395.676,173.836,35.279,156.591
C01431=1061.396,333.341,395.711,173.831,35.274,156.590
C01432=1061.389,333.094,395.746,173.828,35.269,156.589
C01433=1061.383,332.851,395.780,173.824,35.265,156.588
C01434=1061.377,332.609,395.813,173.821,35.260,156.587
C01435=1061.370,332.366,395.847,173.817,35.256,156.586
C01436=1061.364,332.124,395.882,173.813,35.251,156.585
C01437=1061.358,331.882,395.916,173.810,35.247,156.584
C01438=1061.351,331.639,395.950,173.806,35.242,156.583
C01439=1061.345,331.396,395.984,173.803,35.237,156.582
C01440=1061.338,331.154,396.018,173.799,35.233,156.581
C01441=1061.332,330.907,396.053,173.795,35.228,156.580
C01442=1061.326,330.659,396.087,173.792,35.224,156.579
C01443=1061.319,330.412,396.122,173.788,35.219,156.578
C01444=1061.312,330.164,396.156,173.784,35.214,156.577
C01445=1061.305,329.917,396.191,173.781,35.210,156.576
C01446=1061.299,329.669,396.226,173.777,35.205,156.575
C01447=1061.292,329.422,396.259,173.774,35.200,156.574
C01448=1061.285,329.174,396.294,173.769,35.196,156.573
C01449=1061.279,328.926,396.329,173.766,35.192,156.572
C01450=1061.272,328.679,396.363,173.763,35.187,156.571
C01451=1061.265,328.431,396.398,173.759,35.182,156.570
C01452=1061.259,328.184,396.432,173.755,35.178,156.569
C01453=1061.252,327.936,396.466,173.752,35.174,156.568
C01454=1061.245,327.688,396.500,173.748,35.169,156.567
C01455=1061.239,327.440,396.535,173.745,35.165,156.566
C01456=1061.232,327.194,396.569,173.740,35.160,156.565
C01457=1061.225,326.946,396.603,173.737,35.156,156.564
C01458=1061.219,326.698,396.638,173.734,35.151,156.563
C01459=1061.212,326.450,396.671,173.730,35.147,156.562
C01460=1061.206,326.203,396.705,173.727,35.142,156.561
C01461=1061.199,325.955,396.739,173.723,35.138,156.561
C01462=1061.192,325.708,396.774,173.719,35.133,156.560
C01463=1061.186,325.461,396.808,173.716,35.129,156.559
C01464=1061.179,325.213,396.842,173.712,35.124,156.558
C01465=1061.172,324.965,396.877,173.709,35.120,156.557
C01466=1061.166,324.718,396.910,173.706,35.115,156.556
C01467=1061.159,324.470,396.945,173.701,35.111,156.555
C01468=1061.153,324.222,396.979,173.698,35.106,156.554
C01469=1061.146,323.975,397.012,173.695,35.102,156.553
C01470=1061.140,323.727,397.047,173.691,35.097,156.552
C01471=1061.133,323.480,397.080,173.688,35.093,156.551
C01472=1061.127,323.232,397.115,173.685,35.088,156.550
C01473=1061.121,322.984,397.148,173.681,35.084,156.549
C01474=1061.114,322.737,397.182,173.677,35.080,156.548
C01475=1061.108,322.489,397.216,173.673,35.075,156.547
C01476=1061.101,322.242,397.250,173.670,35.071,156.546
C01477=1061.095,321.994,397.284,173.667,35.066,156.545
C01478=1061.088,321.747,397.318,173.663,35.062,156.544
C01479=1061.081,321.499,397.352,173.660,35.058,156.544
C01480=1061.075,321.251,397.385,173.657,35.053,156.543
C01481=1061.069,321.003,397.419,173.653,35.049,156.542
C01482=1061.063,320.756,397.453,173.649,35.044,156.541
C01483=1061.056,320.508,397.487,173.646,35.040,156.540
C01484=1061.050,320.260,397.520,173.642,35.036,156.539
C01485=1061.043,320.013,397.554,173.639,35.031,156.538
C01486=1061.037,319.765,397.588,173.636,35.027,156.537
C01487=1061.030,319.518,397.622,173.632,35.022,156.536
C01488=1061.024,319.270,397.655,173.629,35.018,156.535
C01489=1061.017,319.024,397.689,173.626,35.013,156.534
C01490=1061.011,318.779,397.722,173.622,35.009,156.533
C01491=1061.005,318.534,397.756,173.619,35.005,156.532
C01492=1060.999,318.289,397.789,173.616,35.001,156.531
C01493=1060.992,318.044,397.823,173.612,34.996,156.531
C01494=1060.986,317.798,397.855,173.609,34.992,156.530
C01495=1060.980,317.553,397.889,173.606,34.988,156.529
C01496=1060.974,317.308,397.922,173.602,34.983,156.528
C01497=1060.967,317.060,397.955,173.599,34.979,156.527
C01498=1060.962,316.812,397.989,173.596,34.974,156.526
C01499=1060.955,316.565,398.022,173.592,34.970,156.525
C01500=1060.948,316.317,398.056,173.589,34.966,156.524
C01501=1060.942,316.069,398.089,173.585,34.961,156.523
C01502=1060.936,315.822,398.122,173.581,34.957,156.522
C01503=1060.930,315.574,398.156,173.578,34.953,156.521
C01504=1060.923,315.327,398.190,173.575,34.948,156.520
C01505=1060.918,315.079,398.223,173.571,34.944,156.520
C01506=1060.911,314.832,398.256,173.568,34.940,156.519
C01507=1060.905,314.583,398.290,173.565,34.935,156.518
C01508=1060.899,314.336,398.323,173.562,34.931,156.517
C01509=1060.892,314.089,398.356,173.558,34.926,156.516
C01510=1060.886,313.841,398.390,173.555,34.922,156.515
C01511=1060.879,313.592,398.423,173.552,34.918,156.514
C01512=1060.873,313.345,398.456,173.548,34.914,156.513
C01513=1060.867,313.098,398.489,173.545,34.909,156.512
C01514=1060.860,312.849,398.522,173.542,34.905,156.512
C01515=1060.853,312.602,398.555,173.538,34.901,156.511
C01516=1060.847,312.354,398.588,173.535,34.897,156.510
C01517=1060.840,312.106,398.621,173.532,34.893,156.509
C01518=1060.834,311.858,398.653,173.528,34.889,156.508
C01519=1060.828,311.611,398.686,173.525,34.885,156.507
C01520=1060.821,311.363,398.719,173.522,34.881,156.506
C01521=1060.814,311.116,398.753,173.519,34.877,156.506
C01522=1060.807,310.868,398.785,173.515,34.872,156.505
C01523=1060.801,310.621,398.818,173.512,34.868,156.504
C01524=1060.794,310.373,398.850,173.509,34.864,156.503
C01525=1060.788,310.125,398.883,173.505,34.860,156.502
C01526=1060.781,309.877,398.916,173.502,34.855,156.501
C01527=1060.775,309.630,398.949,173.499,34.851,156.500
C01528=1060.769,309.382,398.982,173.496,34.847,156.499
C01529=1060.762,309.134,399.015,173.492,34.843,156.499
C01530=1060.756,308.885,399.047,173.489,34.839,156.498
C01531=1060.750,308.638,399.080,173.486,34.835,156.497
C01532=1060.743,308.391,399.112,173.482,34.831,156.496
C01533=1060.736,308.143,399.144,173.479,34.827,156.495
C01534=1060.730,307.895,399.177,173.476,34.823,156.494
C01535=1060.723,307.647,399.210,173.474,34.818,156.493
C01536=1060.717,307.400,399.243,173.470,34.814,156.493
C01537=1060.710,307.152,399.276,173.467,34.810,156.492
C01538=1060.704,306.904,399.308,173.464,34.806,156.491
C01539=1060.698,306.656,399.341,173.460,34.802,156.490
C01540=1060.691,306.409,399.373,173.457,34.798,156.489
C01541=1060.685,306.161,399.405,173.454,34.794,156.488
C01542=1060.679,305.914,399.438,173.451,34.790,156.488
C01543=1060.673,305.665,399.470,173.447,34.785,156.487
C01544=1060.666,305.418,399.503,173.444,34.781,156.486
C01545=1060.660,305.174,399.535,173.441,34.777,156.485
C01546=1060.653,304.931,399.567,173.437,34.773,156.484
C01547=1060.647,304.688,399.598,173.435,34.769,156.483
C01548=1060.641,304.444,399.631,173.432,34.765,156.482
C01549=1060.635,304.200,399.663,173.429,34.761,156.482
C01550=1060.629,303.958,399.694,173.425,34.757,156.481
C01551=1060.622,303.714,399.726,173.422,34.753,156.480
C01552=1060.616,303.471,399.758,173.419,34.749,156.479
C01553=1060.610,303.223,399.790,173.416,34.745,156.478
C01554=1060.604,302.975,399.822,173.413,34.741,156.477
C01555=1060.598,302.728,399.855,173.410,34.737,156.477
C01556=1060.591,302.480,399.887,173.407,34.732,156.476
C01557=1060.585,302.232,399.919,173.404,34.728,156.475
C01558=1060.579,301.984,399.951,173.400,34.724,156.474
C01559=1060.572,301.736,399.984,173.397,34.720,156.473
C01560=1060.566,301.488,400.016,173.394,34.716,156.472
C01561=1060.559,301.241,400.048,173.391,34.712,156.472
C01562=1060.553,300.993,400.080,173.388,34.708,156.471
C01563=1060.548,300.745,400.112,173.385,34.704,156.470
C01564=1060.542,300.498,400.145,173.382,34.699,156.469
C01565=1060.536,300.249,400.177,173.378,34.695,156.468
C01566=1060.529,300.002,400.209,173.375,34.691,156.467
C01567=1060.523,299.754,400.241,173.372,34.687,156.466
C01568=1060.517,299.506,400.273,173.370,34.683,156.466
C01569=1060.510,299.258,400.306,173.366,34.679,156.465
C01570=1060.504,299.010,400.337,173.363,34.675,156.464
C01571=1060.498,298.763,400.369,173.360,34.671,156.463
C01572=1060.492,298.515,400.401,173.357,34.667,156.462
C01573=1060.486,298.267,400.433,173.354,34.663,156.461
C01574=1060.479,298.019,400.465,173.351,34.659,156.461
C01575=1060.473,297.771,400.498,173.348,34.655,156.460
C01576=1060.467,297.524,400.529,173.345,34.650,156.459
C01577=1060.461,297.276,400.561,173.341,34.646,156.458
C01578=1060.455,297.028,400.593,173.339,34.642,156.457
C01579=1060.449,296.780,400.625,173.336,34.638,156.456
C01580=1060.442,296.532,400.657,173.333,34.634,156.456
C01581=1060.436,296.285,400.689,173.329,34.630,156.455
C01582=1060.430,296.037,400.720,173.326,34.626,156.454
C01583=1060.424,295.789,400.752,173.324,34.622,156.453
C01584=1060.417,295.541,400.783,173.321,34.618,156.452
C01585=1060.411,295.293,400.816,173.317,34.614,156.452
C01586=1060.404,295.045,400.847,173.314,34.610,156.451
C01587=1060.399,294.797,400.879,173.311,34.606,156.450
C01588=1060.392,294.549,400.910,173.309,34.602,156.449
C01589=1060.385,294.301,400.941,173.305,34.598,156.448
C01590=1060.379,294.053,400.973,173.302,34.594,156.448
C01591=1060.373,293.805,401.005,173.299,34.591,156.447
C01592=1060.367,293.558,401.036,173.297,34.586,156.446
C01593=1060.361,293.310,401.068,173.293,34.582,156.445
C01594=1060.354,293.062,401.099,173.290,34.579,156.444
C01595=1060.347,292.814,401.131,173.287,34.575,156.444
C01596=1060.342,292.566,401.163,173.285,34.570,156.443
C01597=1060.335,292.318,401.193,173.282,34.567,156.442
C01598=1060.329,292.070,401.225,173.278,34.563,156.441
C01599=1060.323,291.822,401.257,173.275,34.559,156.440
C01600=1060.316,291.575,401.288,173.273,34.555,156.440
C01601=1060.310,291.338,401.318,173.270,34.551,156.439
C01602=1060.304,291.103,401.347,173.266,34.547,156.438
C01603=1060.298,290.868,401.377,173.264,34.544,156.437
C01604=1060.293,290.632,401.407,173.261,34.540,156.436
C01605=1060.287,290.395,401.437,173.259,34.536,156.436
C01606=1060.280,290.160,401.466,173.256,34.532,156.435
C01607=1060.274,289.925,401.497,173.252,34.528,156.434
C01608=1060.269,289.689,401.526,173.250,34.525,156.433
C01609=1060.262,289.440,401.557,173.247,34.521,156.433
C01610=1060.256,289.193,401.588,173.244,34.517,156.432
C01611=1060.250,288.945,401.619,173.241,34.513,156.431
C01612=1060.243,288.697,401.650,173.238,34.509,156.430
C01613=1060.238,288.449,401.682,173.235,34.505,156.429
C01614=1060.231,288.201,401.713,173.233,34.502,156.429
C01615=1060.225,287.953,401.744,173.230,34.497,156.428
C01616=1060.218,287.705,401.775,173.226,34.493,156.427
C01617=1060.212,287.457,401.806,173.223,34.490,156.426
C01618=1060.205,287.209,401.837,173.221,34.485,156.426
C01619=1060.199,286.961,401.868,173.218,34.482,156.425
C01620=1060.193,286.714,401.899,173.215,34.478,156.424
C01621=1060.186,286.465,401.930,173.212,34.474,156.423
C01622=1060.180,286.218,401.961,173.209,34.470,156.422
C01623=1060.174,285.969,401.991,173.206,34.466,156.422
C01624=1060.167,285.721,402.023,173.204,34.462,156.421
C01625=1060.161,285.474,402.053,173.201,34.459,156.420
C01626=1060.155,285.226,402.085,173.197,34.454,156.419
C01627=1060.149,284.978,402.115,173.195,34.451,156.419
C01628=1060.142,284.729,402.146,173.192,34.447,156.418
C01629=1060.136,284.481,402.177,173.189,34.443,156.417
C01630=1060.130,284.234,402.207,173.186,34.439,156.416
C01631=1060.123,283.985,402.238,173.183,34.435,156.415
C01632=1060.117,283.738,402.269,173.180,34.431,156.415
C01633=1060.111,283.489,402.300,173.178,34.428,156.414
C01634=1060.105,283.242,402.330,173.175,34.423,156.413
C01635=1060.098,282.994,402.362,173.171,34.420,156.412
C01636=1060.093,282.746,402.392,173.169,34.416,156.412
C01637=1060.086,282.497,402.423,173.166,34.412,156.411
C01638=1060.080,282.250,402.453,173.163,34.408,156.410
C01639=1060.074,282.002,402.485,173.161,34.404,156.409
C01640=1060.068,281.754,402.515,173.157,34.400,156.408
C01641=1060.061,281.505,402.546,173.155,34.397,156.408
C01642=1060.056,281.257,402.576,173.152,34.392,156.407
C01643=1060.049,281.010,402.607,173.149,34.389,156.406
C01644=1060.043,280.762,402.638,173.147,34.385,156.405
C01645=1060.037,280.513,402.669,173.143,34.381,156.405
C01646=1060.031,280.265,402.699,173.141,34.377,156.404
C01647=1060.025,280.018,402.729,173.138,34.373,156.403
C01648=1060.019,279.769,402.760,173.135,34.369,156.402
C01649=1060.012,279.522,402.790,173.133,34.366,156.402
C01650=1060.006,279.273,402.820,173.129,34.361,156.401
C01651=1060.000,279.025,402.851,173.127,34.358,156.400
C01652=1059.993,278.777,402.882,173.124,34.354,156.399
C01653=1059.987,278.529,402.912,173.121,34.350,156.398
C01654=1059.980,278.281,402.942,173.119,34.346,156.398
C01655=1059.974,278.033,402.972,173.116,34.342,156.397
C01656=1059.968,277.784,403.003,173.113,34.339,156.396
C01657=1059.962,277.555,403.031,173.110,34.335,156.395
C01658=1059.956,277.324,403.059,173.108,34.331,156.395
C01659=1059.950,277.094,403.088,173.105,34.328,156.394
C01660=1059.945,276.864,403.115,173.103,34.324,156.393
C01661=1059.940,276.633,403.144,173.100,34.321,156.393
C01662=1059.933,276.403,403.172,173.097,34.317,156.392
C01663=1059.928,276.173,403.200,173.095,34.314,156.391
C01664=1059.922,275.942,403.228,173.092,34.310,156.390
C01665=1059.915,275.694,403.258,173.090,34.306,156.390
C01666=1059.909,275.446,403.288,173.087,34.302,156.389
C01667=1059.903,275.198,403.318,173.084,34.299,156.388
C01668=1059.897,274.950,403.349,173.081,34.295,156.388
C01669=1059.890,274.702,403.378,173.079,34.291,156.387
C01670=1059.885,274.454,403.408,173.076,34.287,156.386
C01671=1059.878,274.205,403.439,173.074,34.284,156.385
C01672=1059.872,273.958,403.469,173.070,34.279,156.384
C01673=1059.866,273.709,403.499,173.067,34.276,156.384
C01674=1059.860,273.461,403.529,173.065,34.272,156.383
C01675=1059.853,273.213,403.559,173.062,34.268,156.382
C01676=1059.848,272.965,403.589,173.060,34.264,156.381
C01677=1059.841,272.717,403.619,173.057,34.260,156.381
C01678=1059.835,272.469,403.649,173.054,34.257,156.380
C01679=1059.828,272.221,403.678,173.051,34.253,156.379
C01680=1059.822,271.972,403.709,173.049,34.249,156.378
C01681=1059.816,271.724,403.739,173.046,34.245,156.378
C01682=1059.810,271.476,403.768,173.044,34.242,156.377
C01683=1059.803,271.229,403.798,173.041,34.237,156.376
C01684=1059.797,270.980,403.828,173.038,34.234,156.375
C01685=1059.791,270.732,403.858,173.035,34.230,156.375
C01686=1059.785,270.484,403.887,173.033,34.226,156.374
C01687=1059.778,270.236,403.918,173.030,34.222,156.373
C01688=1059.772,269.988,403.948,173.028,34.219,156.372
C01689=1059.766,269.740,403.977,173.025,34.215,156.372
C01690=1059.760,269.492,404.007,173.022,34.211,156.371
C01691=1059.753,269.243,404.037,173.019,34.207,156.370
C01692=1059.748,268.994,404.066,173.017,34.203,156.369
C01693=1059.741,268.747,404.096,173.014,34.200,156.369
C01694=1059.736,268.499,404.126,173.012,34.196,156.368
C01695=1059.729,268.251,404.156,173.008,34.192,156.367
C01696=1059.722,268.002,404.185,173.006,34.188,156.366
C01697=1059.717,267.754,404.215,173.003,34.185,156.366
C01698=1059.710,267.506,404.244,173.001,34.180,156.365
C01699=1059.704,267.258,404.273,172.998,34.177,156.364
C01700=1059.698,267.010,404.304,172.996,34.173,156.363
C01701=1059.691,266.761,404.333,172.993,34.170,156.363
C01702=1059.685,266.513,404.362,172.990,34.165,156.362
C01703=1059.680,266.265,404.392,172.988,34.162,156.361
C01704=1059.673,266.017,404.422,172.985,34.158,156.361
C01705=1059.667,265.769,404.451,172.983,34.154,156.360
C01706=1059.660,265.520,404.480,172.980,34.150,156.359
C01707=1059.654,265.272,404.510,172.978,34.147,156.358
C01708=1059.648,265.024,404.539,172.974,34.143,156.357
C01709=1059.642,264.776,404.568,172.972,34.139,156.357
C01710=1059.636,264.528,404.598,172.969,34.135,156.356
C01711=1059.630,264.280,404.627,172.967,34.132,156.355
C01712=1059.623,264.032,404.657,172.965,34.128,156.354
C01713=1059.618,263.803,404.683,172.962,34.124,156.354
C01714=1059.612,263.575,404.711,172.959,34.121,156.353
C01715=1059.606,263.347,404.738,172.957,34.117,156.352
C01716=1059.600,263.118,404.765,172.955,34.114,156.352
C01717=1059.595,262.889,404.792,172.952,34.110,156.351
C01718=1059.588,262.661,404.818,172.950,34.107,156.350
C01719=1059.583,262.432,404.845,172.948,34.103,156.350
C01720=1059.577,262.204,404.872,172.946,34.100,156.349
C01721=1059.571,261.956,404.901,172.942,34.096,156.348
C01722=1059.564,261.708,404.930,172.940,34.093,156.348
C01723=1059.558,261.460,404.959,172.937,34.089,156.347
C01724=1059.552,261.211,404.988,172.935,34.085,156.346
C01725=1059.546,260.963,405.017,172.932,34.082,156.346
C01726=1059.539,260.715,405.046,172.930,34.078,156.345
C01727=1059.533,260.466,405.076,172.928,34.074,156.344
C01728=1059.526,260.218,405.105,172.924,34.070,156.343
C01729=1059.520,259.970,405.134,172.922,34.067,156.343
C01730=1059.513,259.722,405.162,172.919,34.063,156.342
C01731=1059.507,259.474,405.191,172.917,34.059,156.341
C01732=1059.501,259.225,405.220,172.915,34.056,156.340
C01733=1059.495,258.977,405.249,172.912,34.052,156.340
C01734=1059.488,258.729,405.278,172.910,34.048,156.339
C01735=1059.482,258.481,405.307,172.906,34.044,156.338
C01736=1059.476,258.233,405.336,172.904,34.041,156.338
C01737=1059.470,257.985,405.365,172.902,34.037,156.337
C01738=1059.464,257.736,405.393,172.899,34.033,156.336
C01739=1059.457,257.488,405.422,172.897,34.029,156.335
C01740=1059.451,257.239,405.452,172.895,34.026,156.335
C01741=1059.444,256.991,405.481,172.892,34.022,156.334
C01742=1059.438,256.743,405.510,172.889,34.018,156.333
C01743=1059.431,256.494,405.537,172.886,34.014,156.332
C01744=1059.425,256.246,405.566,172.884,34.010,156.332
C01745=1059.419,255.998,405.595,172.882,34.007,156.331
C01746=1059.413,255.749,405.624,172.879,34.003,156.330
C01747=1059.407,255.502,405.652,172.877,34.000,156.330
C01748=1059.401,255.254,405.682,172.875,33.995,156.329
C01749=1059.395,255.005,405.710,172.872,33.992,156.328
C01750=1059.389,254.757,405.739,172.869,33.988,156.327
C01751=1059.383,254.509,405.768,172.867,33.985,156.327
C01752=1059.376,254.260,405.796,172.864,33.980,156.326
C01753=1059.370,254.012,405.825,172.862,33.977,156.325
C01754=1059.363,253.764,405.854,172.860,33.973,156.324
C01755=1059.358,253.515,405.882,172.857,33.969,156.324
C01756=1059.351,253.267,405.911,172.855,33.965,156.323
C01757=1059.345,253.018,405.939,172.852,33.962,156.322
C01758=1059.339,252.770,405.968,172.849,33.958,156.321
C01759=1059.332,252.522,405.996,172.847,33.954,156.321
C01760=1059.326,252.274,406.025,172.845,33.950,156.320
C01761=1059.321,252.026,406.053,172.842,33.946,156.319
C01762=1059.315,251.777,406.082,172.840,33.943,156.319
C01763=1059.309,251.529,406.111,172.838,33.939,156.318
C01764=1059.302,251.281,406.140,172.835,33.935,156.317
C01765=1059.296,251.032,406.168,172.832,33.931,156.316
C01766=1059.289,250.784,406.196,172.830,33.928,156.316
C01767=1059.283,250.535,406.225,172.828,33.924,156.315
C01768=1059.278,250.288,406.253,172.825,33.920,156.314
C01769=1059.272,250.058,406.280,172.823,33.916,156.313
C01770=1059.267,249.829,406.306,172.821,33.913,156.313
C01771=1059.261,249.599,406.332,172.819,33.910,156.312
C01772=1059.255,249.369,406.359,172.817,33.906,156.311
C01773=1059.250,249.140,406.385,172.814,33.902,156.311
C01774=1059.244,248.911,406.411,172.812,33.899,156.310
C01775=1059.238,248.682,406.437,172.810,33.895,156.309
C01776=1059.232,248.452,406.463,172.808,33.892,156.309
C01777=1059.227,248.204,406.491,172.805,33.888,156.308
C01778=1059.221,247.956,406.520,172.803,33.884,156.307
C01779=1059.215,247.707,406.549,172.801,33.881,156.306
C01780=1059.208,247.458,406.576,172.799,33.876,156.306
C01781=1059.203,247.211,406.605,172.795,33.873,156.305
C01782=1059.197,246.962,406.633,172.793,33.869,156.304
C01783=1059.191,246.713,406.662,172.791,33.865,156.303
C01784=1059.185,246.465,406.690,172.789,33.861,156.303
C01785=1059.178,246.218,406.718,172.786,33.858,156.302
C01786=1059.172,245.969,406.746,172.784,33.853,156.301
C01787=1059.166,245.720,406.774,172.782,33.850,156.301
C01788=1059.160,245.472,406.802,172.780,33.846,156.300
C01789=1059.154,245.224,406.830,172.776,33.843,156.299
C01790=1059.148,244.975,406.858,172.774,33.838,156.298
C01791=1059.142,244.726,406.886,172.772,33.835,156.298
C01792=1059.135,244.479,406.915,172.770,33.831,156.297
C01793=1059.129,244.231,406.943,172.767,33.827,156.296
C01794=1059.123,243.982,406.971,172.765,33.823,156.295
C01795=1059.117,243.733,406.999,172.763,33.820,156.295
C01796=1059.111,243.485,407.027,172.761,33.816,156.294
C01797=1059.105,243.237,407.055,172.759,33.812,156.293
C01798=1059.099,242.988,407.083,172.755,33.808,156.292
C01799=1059.092,242.740,407.111,172.753,33.804,156.292
C01800=1059.087,242.492,407.139,172.751,33.801,156.291
C01801=1059.080,242.243,407.166,172.749,33.797,156.290
C01802=1059.074,241.994,407.195,172.747,33.793,156.290
C01803=1059.068,241.747,407.222,172.744,33.789,156.289
C01804=1059.061,241.498,407.250,172.742,33.786,156.288
C01805=1059.056,241.249,407.278,172.740,33.782,156.287
C01806=1059.049,241.001,407.306,172.738,33.778,156.287
C01807=1059.043,240.753,407.333,172.734,33.774,156.286
C01808=1059.037,240.504,407.361,172.732,33.770,156.285
C01809=1059.030,240.255,407.388,172.730,33.767,156.285
